               //calculate crystal orbiting in mm (amplitude-related to crystal center)
               //----------------------------------------------------------------------
               IF ("PAR_MAIN".MCONST_DIA_CAL_P2 > 0.0)   THEN 
                   #xt_orb_mm := 0.5 * ((#max_val_ctr_x_pos - #min_val_ctr_x_pos) / "PAR_MAIN".MCONST_DIA_CAL_P2 * 100.0);     
               END_IF;     

               //set calculation done flag
               //-------------------------
               #orb_calc_done   :=  true;            

               //reset counter 
               //-------------
               #count_msr   :=  0;

           END_IF;

           //set phase related orbiting limit
           //--------------------------------
           IF ("APC".STATUS = "APC".NECK)  THEN
               #up_lim_xt_orb   :=  "PAR_MAIN".MCONST_XT_ORB_LIM_NE;
               #rst_lim_xt_orb  :=  "CNF".RST_LIM_XT_ORB_NE;
           ELSIF ("APC".STATUS = "APC".SHOULDER)  THEN
               #up_lim_xt_orb   :=  "PAR_MAIN".MCONST_XT_ORB_LIM_SH;
               #rst_lim_xt_orb  :=  "CNF".RST_LIM_XT_ORB_SH;
           ELSE 
               #up_lim_xt_orb   :=  "PAR_MAIN".MCONST_XT_ORB_LIM_BY;
               #rst_lim_xt_orb  :=  "CNF".RST_LIM_XT_ORB_BY;
           END_IF;

           //evaluate crystal orbiting
           //-------------------------
           IF #orb_calc_done THEN
               //set orbiting alarm
               //------------------
               IF (#xt_orb_mm > #up_lim_xt_orb) OR "FLT".XT_ORB_ABV_LIM  THEN
                   IF (#set_flt <= 10) THEN      //ten consecutive calculations above limit
                       #set_flt := #set_flt + 1;

                   ELSE
                       //set alarm message
                       //-----------------
                       "FLT".XT_ORB_ABV_LIM  :=  TRUE;

                       //reset orbiting alarm
                       //--------------------
                       IF (#xt_orb_mm < #rst_lim_xt_orb)  THEN
                           IF (#reset_flt <= 30) THEN   //thirty consecutive calculations below limit
                               #reset_flt := #reset_flt + 1;

                           ELSE
                               //reset alarm message and flags
                               //-----------------------------
                               "FLT".XT_ORB_ABV_LIM  :=  FALSE;
                               #set_flt             :=  0;
                               #reset_flt           :=  0;
                           END_IF;
                       ELSE 
                           #reset_flt := 0;
                       END_IF;
                   END_IF;
               ELSE
                   #set_flt := 0;
               END_IF;
           END_IF;

       //crystal orbiting is deactivated
       //-------------------------------                          
       ELSE
           "FLT".XT_ORB_ABV_LIM  :=  FALSE;
           #xt_orb_mm           :=  0.0;
           #count_msr           :=  0;
           #set_flt             :=  0;
           #reset_flt           :=  0;
       END_IF;

       //set display value crystal orbiting
       //----------------------------------
       "DIS".ACT_XT_ORB  :=  #xt_orb_mm;
END_FUNCTION_BLOCK

FUNCTION_BLOCK "BM_MLT_LVL_MON"   // FB93, SCL
{ S7_Optimized_Access := 'FALSE' }
VERSION : 0.0
// --------------------------------------------------------------------------------
//     program     :    BM_MLT_LVL_MON
//     description :    melt level monitoring       
//     name        :    G. Eibelsh鋟ser
//     date        :    28.10.2009
// 
//     revision    :
//     name        :
//     date        :    
//                     (c)PVATepla AG
//     --------------------------------------------------------------------------------
   VAR
      ctl_mlt_drift_on : Bool;
      ctl_mlt_drift_on_dly : Int;
      cal_mlt_lvl_mm : Real;
      ini_mlt_lvl_mm : Real;
   END_VAR
BEGIN


       //monitoring of melt level in phases IDLE and BODY
       //------------------------------------------------
       IF ("APC".STATUS = "APC".IDLE) OR ("APC".STATUS = "APC".BODY) THEN 
           //calibrate melt level in unit mm
           //-------------------------------
           #cal_mlt_lvl_mm  :=  "AV".AVG_PRD_2_CTR_Y * "PAR_MAIN".MCONST_MLT_LVL_CAL;   //cal factor in unit mm/pixel

           //camera is on and circle sensor is selected
           //------------------------------------------
           IF "LT".CAM_ISP_ON AND ("AV".ACT_DVT_PRD_NO = 2.0) THEN 

               //automatic reset of melt level value in phase BODY
               //-------------------------------------------------
               IF ("APC".STATUS = "APC".BODY) AND ("AV".ACT_XT_LEN < "PAR_MAIN".BY_XT_LGH_MLT_LVL_RST) THEN     //actual crystal length below or equal activation length
                   "AV".ACT_MLT_LVL      :=  0.0;
                   #ini_mlt_lvl_mm      :=  #cal_mlt_lvl_mm;
                   #ctl_mlt_drift_on    :=  false;                          //disable melt drift control loop

               //melt level calculation
               //----------------------
               ELSE                                                        
                   IF ("APC".AUTOMATIC AND ("APC".STATUS = "APC".BODY) AND (REAL_TO_INT("PAR_MAIN".BY_CTL_MLT_DRIFT_ON) = 1) AND NOT "SY".CTL_OFFS_SPEED_ON) THEN  //crystal length exceeded activation length
                       #ctl_mlt_drift_on    :=  true;                       //enable melt drift control loop
                   ELSE
                       #ctl_mlt_drift_on    :=  false;                      //disable melt drift control loop
                   END_IF;

                   //stereo camera mode active
                   //-------------------------
                   IF (("CNF".ACT_DVC_CNF AND 2#0000_0000_0000_1000_0000_0000_0000_0000) = 2#0000_0000_0000_1000_0000_0000_0000_0000) THEN 
                       "AV".ACT_MLT_LVL   :=  "AV".S_CAM_AVG_MLT_LVL_CHG;  //pos. value >> melt gap gets larger, neg. value >> melt gap gets smaller

                   //single camera mode active
                   //-------------------------
                   ELSE 
                       //manual reset of melt level value
                       //--------------------------------
                       IF      NOT "APC".AUTOMATIC               //manual mode
                           OR      "SY".CTL_CR_SPD_COF_SMI       //semi mode crucible speed coeffizient
                           OR      "SY".CTL_MLT_LVL_SMI THEN     //semi mode crucible speed

                           IF "KYD".RST_MLT_LVL THEN
                               #ctl_mlt_drift_on    :=  false;                  //disable melt drift control loop while reseting 
                               #ini_mlt_lvl_mm      :=  #cal_mlt_lvl_mm;
                               "LT".RST_MLT_LVL      :=  TRUE;
                           END_IF;                
                       END_IF;
                       //calculation of actual melt level
                       //--------------------------------
                       "AV".ACT_MLT_LVL   :=  #cal_mlt_lvl_mm - #ini_mlt_lvl_mm;   //pos. value >> melt gap gets larger, neg. value >> melt gap gets smaller
                   END_IF;
               END_IF;

               //alarm setting in phase BODY
               //---------------------------
               IF ("APC".STATUS = "APC".BODY) AND ("PAR_MAIN".LIM_MLT_LVL_DEV >= 0.1) THEN   
                   //set alarm messages when distance from melt to funnel is too large
                   //-----------------------------------------------------------------
                   IF ("AV".ACT_MLT_LVL < "PAR_MAIN".LIM_MLT_LVL_DEV * 0.5) THEN
                       "FLT".DST_MLT_FNL_LRG :=  FALSE;

                   ELSIF ("AV".ACT_MLT_LVL > "PAR_MAIN".LIM_MLT_LVL_DEV) THEN
                       "FLT".DST_MLT_FNL_LRG :=  TRUE;

                   END_IF;

                   //set alarm messages when distance from melt to funnel is too small
                   //-----------------------------------------------------------------
                   IF ("AV".ACT_MLT_LVL > ("PAR_MAIN".LIM_MLT_LVL_DEV * (-0.5))) THEN  
                       "FLT".DST_MLT_FNL_SML :=  FALSE;

                   ELSIF ("AV".ACT_MLT_LVL < ("PAR_MAIN".LIM_MLT_LVL_DEV * (-1.0))) THEN  
                       "FLT".DST_MLT_FNL_SML :=  TRUE;

                   END_IF;

               ELSE
                   "FLT".DST_MLT_FNL_LRG :=  FALSE;
                   "FLT".DST_MLT_FNL_SML :=  FALSE;

               END_IF;

           //reset variables and alarms
           //--------------------------
           ELSE
               "AV".ACT_MLT_LVL      :=  0.0;
               #ini_mlt_lvl_mm      :=  #cal_mlt_lvl_mm;
               #ctl_mlt_drift_on    :=  false;                          //disable melt drift control loop
               "FLT".DST_MLT_FNL_LRG :=  FALSE;
               "FLT".DST_MLT_FNL_SML :=  FALSE;

           END_IF;

       ELSE
           //reset variables and alarms
           //--------------------------
           "AV".ACT_MLT_LVL      :=  0.0;
           #ctl_mlt_drift_on    :=  false;                          //disable melt drift control loop
           "FLT".DST_MLT_FNL_LRG :=  FALSE;
           "FLT".DST_MLT_FNL_SML :=  FALSE;

       END_IF;

       //enable control loop melt level drift
       //------------------------------------
       "DC".CTL_MLT_DRIFT_ON :=  "SysOndelay"( DIN     := #ctl_mlt_drift_on,
                                           SetTime := 30,                      // setp. time
                                           ActTime := #ctl_mlt_drift_on_dly,    // act. time
                                           Tick    := "SysTick1s");              // timebase (1s)

       //write display value of actual melt level
       //----------------------------------------
       "DIS".ACT_MLT_LVL  :=  "AV".ACT_MLT_LVL;
END_FUNCTION_BLOCK

FUNCTION_BLOCK "BM_MLT_VIB_MON"   // FB94, SCL
{ S7_Optimized_Access := 'FALSE' }
VERSION : 0.0
// --------------------------------------------------------------------------------
//     program     :    BM_MLT_VIB_MON
//     description :    melt vibration monitoring
//     name        :    G. Eibelsh鋟ser
//     date        :    01.09.2011
// 
//     revision    :
//     name        :
//     date        :    
//                     (c)PVA Tepla AG
//     --------------------------------------------------------------------------------
   VAR
      melt_vib_mon : Bool;
      store_mlt_vib_raw : Bool;
      cnt_msr : Int;
      cnt_msr_raw : Int;
      cnt_1s : Int;
      mlt_vib_dist : Array[1..300] of Real;
      mlt_vib_dist_raw : Array[1..100] of Real;
      min_mlt_vib_dist : Real;
      max_mlt_vib_dist : Real;
      mlt_vib_dist_pix : Real;
   END_VAR
   VAR CONSTANT
      amt_of_msr : Int := 10;
      amt_msr_raw : Int := 100;
   END_VAR
BEGIN


       //activate melt vibration monitoring
       //----------------------------------
       #melt_vib_mon := "LT".CAM_ISP_ON;

       //melt vibration monitoring is activated
       //--------------------------------------                          
       IF #melt_vib_mon  THEN

           //read sensor vibration distance
           //------------------------------  
           IF "DV".NEW_MSR_TEL_RECV THEN                         //new measurement telegram received
               #cnt_msr                 := #cnt_msr + 1;         //increase counter variable after each measurement
               #mlt_vib_dist[#cnt_msr]   := "AV".ACT_MLT_VIB_DIST; //store melt vibration distance in array variable
           END_IF;

           //evaluate measurement points
           //---------------------------
           IF (#cnt_msr >= #amt_of_msr) THEN

               //call min max detection
               //----------------------
               "CM_MIN_MAX"( record      := #mlt_vib_dist,
                           amt_of_val  := #amt_of_msr,
                           min_value   := #min_mlt_vib_dist, 
                           max_value   := #max_mlt_vib_dist);

               //calculate difference between min and max value
               //----------------------------------------------
               #mlt_vib_dist_pix := #max_mlt_vib_dist - #min_mlt_vib_dist;     

               //reset counter 
               //-------------
               #cnt_msr   :=  0;
           END_IF;    

           //store raw values of melt vibration sensor
           //-----------------------------------------
           IF "LT".MSR_MLT_VIB_ON THEN 
               IF #store_mlt_vib_raw THEN

                   //read sensor vibration distance
                   //------------------------------  
                   IF "DV".NEW_MSR_TEL_RECV THEN                                     //new measurement telegram received
                       #cnt_msr_raw                   := #cnt_msr_raw + 1;           //increase counter variable after each measurement
                       #mlt_vib_dist_raw[#cnt_msr_raw] := "AV".ACT_MLT_VIB_DIST;       //store melt vibration distance in array variable
                   END_IF;
                   //stop storage after selected amount of values
                   //--------------------------------------------
                   IF (#cnt_msr_raw >= #amt_msr_raw) THEN 
                       #store_mlt_vib_raw   :=  false;
                   END_IF;
               END_IF;

               //write raw values in display variables in 1 second intervall
               //-----------------------------------------------------------
               IF (#cnt_msr_raw >= 1) THEN 
                   IF "SysTick1s" THEN
                       IF (#cnt_1s >= #amt_msr_raw) THEN                         //stop writing after selected amount of seconds
                           "LT".MSR_MLT_VIB_ON   :=  FALSE;
                       ELSE
                           #cnt_1s              := #cnt_1s + 1;                  //increase 1 second counter
                           "DIS".ACT_MLT_VIB_RAW := #mlt_vib_dist_raw[#cnt_1s];    //write display value
                       END_IF;
                   END_IF;
               END_IF;

           //reset variables
           //---------------
           ELSE     
               #cnt_msr_raw         :=  0;
               #cnt_1s              :=  0;
               "DIS".ACT_MLT_VIB_RAW :=  0.0;
           END_IF;

           //activate storage of raw values from melt vibration sensor
           //---------------------------------------------------------
           IF "KYD".MSR_MLT_VIB_ON AND NOT "LT".MSR_MLT_VIB_ON THEN
               "LT".MSR_MLT_VIB_ON   :=  TRUE;
               #store_mlt_vib_raw   :=  true;
           END_IF;

       //reset variables
       //---------------
       ELSE    
           #cnt_msr             :=  0;
           #cnt_msr_raw         :=  0;
           #cnt_1s              :=  0;
           #mlt_vib_dist_pix    :=  0.0;
           "DIS".ACT_MLT_VIB_RAW :=  0.0;
           "LT".MSR_MLT_VIB_ON   :=  FALSE;
           #store_mlt_vib_raw   :=  false;
       END_IF;

       //write display value of actual melt vibration
       //--------------------------------------------
       "DIS".ACT_MLT_VIB :=  #mlt_vib_dist_pix;
END_FUNCTION_BLOCK

FUNCTION_BLOCK "BM_S_CAM_EVAL"   // FB99, SCL
{ S7_Optimized_Access := 'FALSE' }
VERSION : 0.0
// --------------------------------------------------------------------------------
//     program     :    BM_S_CAM_EVAL
//     description :    stereo camera evaluation  
//     name        :    G. Eibelsh鋟ser
//     date        :    20.08.2019
//        
//     revision    :   
//     name        :   
//     date        :   
//        
//                     (c)PVA Tepla AG
//     --------------------------------------------------------------------------------
   VAR
      s_cam_1_init_rad_pt : Real;
      s_cam_2_init_rad_pt : Real;
      s_cam_last_cf_dia : Real;
      s_cam_act_mlt_lvl_chg : Real;
      ini_mlt_lvl_inp : Real;
   END_VAR
   VAR_TEMP
      term_1 : Real;
      term_2 : Real;
      term_3 : Real;
      term_4 : Real;
      delta_x1 : Real;
      delta_x2 : Real;
      delta_r : Real;
      delta_h : Real;
   END_VAR
BEGIN


       //calculate trigonometric terms (angle in radiant)
       //------------------------------------------------
       #term_1  :=  SIN("CNF".PI * ("PAR_MAIN".MCONST_ANG_OF_PLX_SCAM - "CNF".S_CAM_ANG_BETA /2) /180);
       #term_2  :=  SIN("CNF".PI * ("PAR_MAIN".MCONST_ANG_OF_PLX_SCAM + "CNF".S_CAM_ANG_BETA /2) /180);
       #term_3  :=  COS("CNF".PI * ("PAR_MAIN".MCONST_ANG_OF_PLX_SCAM - "CNF".S_CAM_ANG_BETA /2) /180);
       #term_4  :=  COS("CNF".PI * ("PAR_MAIN".MCONST_ANG_OF_PLX_SCAM + "CNF".S_CAM_ANG_BETA /2) /180);

       //store initial radius point during circle fit
       //--------------------------------------------
       IF  NOT "DV".S_CAM_RAD_RT_ACTV   THEN
           #s_cam_1_init_rad_pt :=  "AV".S_CAM_1_AVG_RAD_PT;  
           #s_cam_2_init_rad_pt :=  "AV".S_CAM_2_AVG_RAD_PT;

       ELSE 
           //calculate radius from measured points of both cameras
           //-----------------------------------------------------
           #delta_x1 :=  #s_cam_1_init_rad_pt - "AV".S_CAM_1_AVG_RAD_PT;
           #delta_x2 :=  #s_cam_2_init_rad_pt - "AV".S_CAM_2_AVG_RAD_PT;

           //calculate radius of crystal from both camera inputs
           //--------------------------------------------------- 
           #delta_r := (#delta_x2 / #term_1 - #delta_x1 / #term_2) / (#term_3 / #term_1 - #term_4 / #term_2);

           //calculate melt level change from both camera inputs
           //--------------------------------------------------- 
           #delta_h := (#delta_x2 / #term_3 - #delta_x1 / #term_4) / (#term_1 / #term_3 - #term_2 / #term_4);

       END_IF;

       //write diameter and melt level variable
       //--------------------------------------
       //reset diamter and melt level change when camera off or diameter measuement mode not selected
       //--------------------------------------------------------------------------------------------
       IF NOT ("LT".CAM_ISP_ON AND "LT".CAM_DIA) THEN
           "AV".S_CAM_ACT_XT_DIA     :=  0.0;
           #s_cam_act_mlt_lvl_chg   :=  0.0;
       //radius point evaluation
       //-----------------------
       ELSIF "DV".S_CAM_RAD_RT_ACTV  THEN
           "AV".S_CAM_ACT_XT_DIA     :=  #s_cam_last_cf_dia + #delta_r * 2 / "PAR_MAIN".MCONST_CAL_RAD_PT_SCAM * 100 - "AC".XT_MENISCUS;   //unit of diameter calibration factor is pix/100mm
           //melt level change
           //-----------------
           #s_cam_act_mlt_lvl_chg   :=  #delta_h / "PAR_MAIN".MCONST_CAL_MLT_LVL_SCAM *(-1);   //unit of melt level calibration factor is pix/mm - neg. value >> reduced gap, pos. val. >> increased gap

       //circle fit evaluation
       //---------------------
       ELSE
           "AV".S_CAM_ACT_XT_DIA     :=  "AV".S_CAM_1_ACT_DIA_CF / "PAR_MAIN".MCONST_CAL_CF_SCAM * 100 - "AC".XT_MENISCUS;     //unit of diameter calibration factor is pix/100mm
           #s_cam_last_cf_dia       :=  "AV".S_CAM_ACT_XT_DIA + "AC".XT_MENISCUS;
           #s_cam_act_mlt_lvl_chg   :=  0.0;
       END_IF;

       //set point evaluation type - radius point detection or circle fit
       //----------------------------------------------------------------
       IF ("APC".STATUS <= "APC".NECK) THEN
           "DV".S_CAM_RAD_RT_ACTV   :=  FALSE;
       ELSIF ((("APC".STATUS = "APC".SHOULDER) AND ("AV".S_CAM_AVG_XT_DIA > "PAR_MAIN".MCONST_CF_TO_RAD_PT_SCAM)) OR ("APC".STATUS = "APC".BODY)) THEN
           "DV".S_CAM_RAD_RT_ACTV   :=  TRUE;
       END_IF;

       //manual reset of melt level value
       //--------------------------------
       IF ("KYD".RST_MLT_LVL AND NOT "LT".CTL_MLT_DRIFT_ON) THEN                   //melt drift control must be off
           "LT".RST_MLT_LVL := "KYD".RST_MLT_LVL AND NOT "LT".CTL_MLT_DRIFT_ON;      //reset in cm_loops
       END_IF;

       //melt level change calc in body after minimum length
       //---------------------------------------------------
       IF ("APC".STATUS = "APC".BODY) AND ("AV".ACT_XT_LEN >= "PAR_MAIN".BY_XT_LGH_MLT_LVL_RST) AND NOT "LT".RST_MLT_LVL THEN
           "AV".S_CAM_ACT_MLT_LVL_CHG    :=  #ini_mlt_lvl_inp - #s_cam_act_mlt_lvl_chg;
       //reset melt level change values
       //------------------------------
       ELSE
           #ini_mlt_lvl_inp             :=  #s_cam_act_mlt_lvl_chg;
           "AV".S_CAM_ACT_MLT_LVL_CHG    :=  0.0;
       END_IF;
END_FUNCTION_BLOCK

FUNCTION_BLOCK "BM_CALL_CAM"   // FB100, SCL
{ S7_Optimized_Access := 'FALSE' }
VERSION : 0.0
// --------------------------------------------------------------------------------
//     program     :    BM_CALL_CAM
//     description :    call camera modules 
//     name        :    G. Eibelsh鋟ser
//     date        :    03.05.2010
// 
//     revision    :    
//     name        :    
//     date        :    
//                     (c)PVA Tepla AG
//     --------------------------------------------------------------------------------
   VAR
      CAM_1_COM : "BM_CAM_COM";
      CAM_1_RSP : "BM_CAM_RSP";
      CAM_CONTROL : "BM_CAM_CONTROL";
      cam_1_req_msr : Bool;
      cam_1_send_req : Bool;
      cam_2_send_req : Bool;
      cam_1_send_done : Bool;
      cam_1_send_err : Bool;
      cam_1_recv_ndr : Bool;
      cam_1_recv_err : Bool;
      cam_1_eval_data : Bool;
      cam_1_data_str_recv : Bool;
      enb_dia_eval : Bool;
      no_ctr_fnd : Bool;
      wait_for_rsp : Bool;
      phase_shift : Bool;
      itl_cam_flt : Bool;
      xt_rot_cam_trg_prv : Bool;
      kyd_ext_acq_trg_busy : Bool;
      do_fac_shot_with_dly : Bool;
      sta_tme_trig_fac_shot : Bool;
      send_fac_shot_msg : Bool;
      cam_1_recv_len : Int;
      retval_blk : Int;
      i : Int;
      "m" : Int;
      n : Int;
      no_ctr_fnd_dly : Int;
      wait_for_rsp_dly : Int;
      itl_cam_flt_dly : Int;
      cam_no_ctr_fnd_dly : Int;
      mlt_amt_of_blobs : Int;
      apc_status : Int;
      dly_cnt : Int;
      acq_cnt : Int;
      next_fac_pic : Int;   // 0= fac1 1= fac2 2= fac3 3= fac4
      dly_fac_shot : Int;
      dly_cnt_fac_shot : DInt;   // added for single shot of facet
      cam_1_send_stat : Word;
      cam_1_recv_stat : Word;
      dip_int_on_line : Real;
      dia_cir_fit : Real;
      dia_cir_fit_old : Real;
      ctr_x_crd_cir_fit : Real;
      ctr_y_crd_cir_fit : Real;
      mlt_vib_dist : Real;
      dia_line_msr : Real;
      dia_pts_incl : Real;
      dia_cal_cir_fit : Real;
      dia_cal_pts_incl : Real;
      ctr_x_crd_cal_cir_fit : Real;
      ctr_y_crd_cal_cir_fit : Real;
      s_cam_delta_r : Real;   // added for stereo camera test
      s_cam_delta_h : Real;
      dia_circ_fit_x1 : Real;
      dia_circ_fit_x2 : Real;
      act_radius_x1 : Real;
      act_radius_x2 : Real;
      ctr_x_circ_fit_s_cam1 : Real;
      ctr_y_circ_fit_s_cam1 : Real;
      ctr_x_circ_fit_s_cam2 : Real;
      ctr_y_circ_fit_s_cam2 : Real;
      plc_to_sherlock : String[254];
   END_VAR
   VAR_TEMP
      rot_trg_acq_req : Bool;
      ms_btw_fct : Real;
   END_VAR
   VAR CONSTANT
      max_pix_intensity : Int := 255;
      amt_of_fct : Int := 4;   // amount of facettes
      min_xt_rot : Int := 2;   // minimum crystal rotation for external acqisition trigger
      time_base : Real := 60000.0;   // minute in ms
      time_trig_fac : DInt := 180000;   // all 3 min
   END_VAR
BEGIN


       //call camera control 
       //-------------------
       #CAM_CONTROL();

       //switch external acquisition trigger on/off
       //------------------------------------------
       IF "LT".XT_ROT_OFF OR ("KYA".SET_XT_ROT < #min_xt_rot) THEN 
           "LT".EXT_ACQ_TRG_ON   :=  FALSE;
       ELSE
           "SM_POS_EDGE"(input   :=  "KYD".EXT_ACQ_TRG,         //button external acquisiton trigger on/off
                       busy    :=  #kyd_ext_acq_trg_busy,
                       output  :=  "LT".EXT_ACQ_TRG_ON);
       END_IF;

       //calculate time between two facettes in ms
       //-----------------------------------------
       IF "LT".EXT_ACQ_TRG_ON THEN 
           #ms_btw_fct :=  #time_base / "KYA".SET_XT_ROT /#amt_of_fct;
       ELSE
           #ms_btw_fct :=  0.0;
       END_IF;

       //reset delay time with positive edge of rotation indexer
       //-------------------------------------------------------
       IF "PDI".XT_ROT_CAM_TRG AND NOT #xt_rot_cam_trg_prv OR NOT "LT".EXT_ACQ_TRG_ON THEN
           #dly_cnt     :=  0;
           #acq_cnt     :=  0;

       //increase delay time with cycle time of previous cycle
       //-----------------------------------------------------
       ELSE
           #dly_cnt :=  #dly_cnt + "SY".OB1_PREV_CYCLE;
       END_IF;

       //For the facet pic
       IF "LT".EXT_ACQ_TRG_ON AND "LT".CAM_ISP_ON THEN
           #dly_cnt_fac_shot:= #dly_cnt_fac_shot + "SY".OB1_PREV_CYCLE;
           IF #dly_cnt_fac_shot > #time_trig_fac THEN
               #next_fac_pic:= #next_fac_pic + 1;
               IF #next_fac_pic > 3 THEN
                   #next_fac_pic:=0;
               END_IF;
               #dly_cnt_fac_shot:=0;
               #do_fac_shot_with_dly:=TRUE;
           END_IF;

       ELSE
           #dly_cnt_fac_shot:= 0;
           #next_fac_pic:=-1;
           #do_fac_shot_with_dly:=FALSE;
           #sta_tme_trig_fac_shot:=FALSE;
           #send_fac_shot_msg:=FALSE;
       END_IF;

       //store status of rotation indexer of current cycle
       //-------------------------------------------------
       #xt_rot_cam_trg_prv  :=  "PDI".XT_ROT_CAM_TRG;

       //set rotation triggered acquisition request when delay time over
       //---------------------------------------------------------------
       IF ("LT".EXT_ACQ_TRG_ON AND (#dly_cnt >= (REAL_TO_INT("KYA".CAM_ACQ_DLY) + (#acq_cnt * #ms_btw_fct)))) THEN
           //When the fac should be shot after 3 min then look for the right fac and then do the pic
           IF #do_fac_shot_with_dly AND (#next_fac_pic = #acq_cnt) THEN
               #do_fac_shot_with_dly:=FALSE;
               #sta_tme_trig_fac_shot:=TRUE;
           END_IF;
           #rot_trg_acq_req :=  true;
           #acq_cnt         :=  #acq_cnt + 1;
       ELSE
           #rot_trg_acq_req := false;
       END_IF;

       //If the fac is been triggert by the area between the facettes a time of 1/2 the 1/4 rot time
       IF #sta_tme_trig_fac_shot THEN
           #dly_fac_shot:= #dly_fac_shot + "SY".OB1_PREV_CYCLE;
           IF #dly_fac_shot >= #ms_btw_fct/2 THEN
               #send_fac_shot_msg:=TRUE;
               #dly_fac_shot:=0;
               #sta_tme_trig_fac_shot:=FALSE;
           END_IF;
       END_IF;

       //set camera measurement request
       //------------------------------
       IF "LT".CAM_ISP_ON THEN
           IF "LT".EXT_ACQ_TRG_ON  THEN                  //external acquisition trigger active
               IF #rot_trg_acq_req THEN                 //triggered from rotation indexer, one acquisiton per rotation
                   #cam_1_req_msr :=  true;
               END_IF;
           ELSIF ("CNF".IMG_AQI_TRG = 100)  THEN
               IF "SysTick100ms" THEN                    //10Hz
                   #cam_1_req_msr :=  true;
               END_IF;
           ELSIF ("CNF".IMG_AQI_TRG = 200)  THEN
               IF "SysTick200ms" THEN                    //5Hz
                   #cam_1_req_msr :=  true;
               END_IF;
           ELSIF ("CNF".IMG_AQI_TRG = 500)  THEN
               IF "SysTick500ms" THEN                    //2Hz
                   #cam_1_req_msr :=  true;
               END_IF;
           ELSIF ("CNF".IMG_AQI_TRG = 1000)  THEN
               IF "SysTick1s" THEN                       //1Hz
                   #cam_1_req_msr :=  true;
               END_IF;
           END_IF;
       ELSE        
           #cam_1_req_msr :=  false;    //reset measurement request
       END_IF;

       //write send string
       //-----------------
       IF (#CAM_1_COM.O_SEND_STAT = 16#0000) AND NOT #wait_for_rsp   THEN       //no send task running and response on last request received

           //switch on image acquisition
           //---------------------------
           IF #CAM_CONTROL.O_ACQ_ON THEN
               #plc_to_sherlock             :=  'acq_on_';                          //set data 
               #cam_1_send_req              :=  true;                               //set send request
               #wait_for_rsp                :=  true;                               //wait for response
               #CAM_CONTROL.O_ACQ_ON        :=  FALSE;

           //switch off image acquisition
           //---------------------------
           ELSIF #CAM_CONTROL.O_ACQ_OFF THEN
               #plc_to_sherlock             :=  'acq_off';                          //set data 
               #cam_1_send_req              :=  true;                               //set send request
               #wait_for_rsp                :=  true;                               //wait for response
               #CAM_CONTROL.O_ACQ_OFF       :=  FALSE;

           //switch on relative threshold
           //----------------------------
           ELSIF #CAM_CONTROL.O_THR_REL_ON THEN
               #plc_to_sherlock             :=  'thr_rel';                          //set data 
               #cam_1_send_req              :=  true;                               //set send request
               #wait_for_rsp                :=  true;                               //wait for response
               #CAM_CONTROL.O_THR_REL_ON    :=  FALSE;

           //switch switch on absolute threshold
           //-----------------------------------
           ELSIF #CAM_CONTROL.O_THR_ABS_ON THEN
               #plc_to_sherlock             :=  'thr_abs';                          //set data 
               #cam_1_send_req              :=  true;                               //set send request
               #wait_for_rsp                :=  true;                               //wait for response
               #CAM_CONTROL.O_THR_ABS_ON    :=  FALSE;

           //switch on neck measurement mode for stereo cameras     - added for stereo camera test
           //--------------------------------------------------
           ELSIF #CAM_CONTROL.O_CF_EVAL THEN
               #plc_to_sherlock             :=  'cfit_ne';                          //set data 
               #cam_1_send_req              :=  true;                               //set send request
               #wait_for_rsp                :=  true;                               //wait for response
               #CAM_CONTROL.O_CF_EVAL       :=  FALSE;

           //switch off neck measurement mode for stereo cameras
           //---------------------------------------------------
           ELSIF #CAM_CONTROL.O_RAD_PT_EVAL THEN
               #plc_to_sherlock             :=  'pfit_sb';                          //set data 
               #cam_1_send_req              :=  true;                               //set send request
               #wait_for_rsp                :=  true;                               //wait for response
               #CAM_CONTROL.O_RAD_PT_EVAL   :=  FALSE;

           //ROI coordinate change is requested
           //----------------------------------
           ELSIF #CAM_CONTROL.O_NEW_ROI_CRD    THEN
               #plc_to_sherlock             BLKMOV  #CAM_CONTROL.O_ROI_CRD_STRG;         //set data 
               #cam_1_send_req              :=  true;                               //set send request
               #wait_for_rsp                :=  true;                               //wait for response
               #CAM_CONTROL.O_NEW_ROI_CRD   :=  FALSE;                              //reset flag new ROI coordinates

           //ROI threshold change is requested
           //---------------------------------
           ELSIF #CAM_CONTROL.O_NEW_ROI_THR  THEN                                   //set data
               #plc_to_sherlock             BLKMOV  #CAM_CONTROL.O_ROI_THR_STRG;
               #cam_1_send_req              :=  true;                               //set send request
               #wait_for_rsp                :=  true;                               //wait for response
               #CAM_CONTROL.O_NEW_ROI_THR   :=  FALSE;                              //reset flag new ROI coordinates

           //ROI threshold 2 change is requested
           //---------------------------------
           ELSIF #CAM_CONTROL.O_NEW_ROI_THR_2  THEN                                 //set data from camera 2
               #plc_to_sherlock             BLKMOV  #CAM_CONTROL.O_ROI_THR_STRG_2;
               #cam_1_send_req              :=  true;                               //set send request
               #wait_for_rsp                :=  true;                               //wait for response
               #CAM_CONTROL.O_NEW_ROI_THR_2 :=  FALSE;                              //reset flag new ROI coordinates

           //do a single pic of the facet    
           ELSIF #send_fac_shot_msg THEN
               CASE #next_fac_pic OF 
                   0:#plc_to_sherlock       :=  'pic_fac1';                          //set data                    
                   1:#plc_to_sherlock       :=  'pic_fac2';                          //set data 
                   2:#plc_to_sherlock       :=  'pic_fac3';                          //set data 
                   3:#plc_to_sherlock       :=  'pic_fac4';                          //set data 
               END_CASE;
               #cam_1_send_req              :=  true;                               //set send request
               #wait_for_rsp                :=  true;                               //wait for response
               #send_fac_shot_msg           :=  FALSE;                              //reset flag new ROI coordinates

           //cyclic measurement is requested
           //-------------------------------
           ELSIF #cam_1_req_msr THEN     
               //set plc command string
               //----------------------
               IF "LT".CAM_MLT THEN
                   #plc_to_sherlock    :='mlt_msr';        //melt detection measurement
               ELSIF "LT".CAM_DIP THEN
                   #plc_to_sherlock    :='dip_msr';        //dipping detection
               ELSIF "LT".CAM_DIA THEN
                   IF "LT".CAM_PRD_1_SEL THEN
                       #plc_to_sherlock    :='dia_rec';    //diameter measurement with rectangle ROI
                   ELSIF "LT".CAM_PRD_2_SEL THEN 
                       #plc_to_sherlock    :='dia_msr';    //diameter measurement with segmented circle ROI
                   END_IF;
               END_IF;

               #cam_1_send_req  :=  true;               //set send request
               #wait_for_rsp    :=  true;               //wait for response

               //reset measurement request
               //-------------------------
               #cam_1_req_msr       :=  false;          

           END_IF;    
       END_IF;

       //call TCP/IP communication of sherlock
       //-------------------------------------
       #CAM_1_COM  (IO_SEND_REQ         :=  #cam_1_send_req,
                   IO_DATA_STR_RECV    :=  #cam_1_data_str_recv,
                   I_SEND_CON_ID       :=  "CNF".CAM_1_CON_ID_SEND,
                   I_RECV_CON_ID       :=  "CNF".CAM_1_CON_ID_RECV,
                   I_CP_ADR            :=  "CNF".CP_LADDR,
                   I_DATA_STRING       BLKMOV  #plc_to_sherlock);

                   #cam_1_send_done     :=  #CAM_1_COM.O_SEND_DONE;
                   #cam_1_send_err      :=  #CAM_1_COM.O_SEND_ERR;
                   #cam_1_recv_ndr      :=  #CAM_1_COM.O_RECV_NDR;
                   #cam_1_recv_err      :=  #CAM_1_COM.O_RECV_ERR;
                   #cam_1_recv_len      :=  #CAM_1_COM.O_RECV_LEN;

                   #cam_1_send_stat     :=  #CAM_1_COM.O_SEND_STAT;
                   #cam_1_recv_stat     :=  #CAM_1_COM.O_RECV_STAT;

       "DV".NEW_MSR_TEL_RECV :=  FALSE;  //reset new measurement telegram variable            

       //move data from receive DB to data DB
       //------------------------------------
       IF #cam_1_data_str_recv THEN
           #retval_blk          :=  BLKMOV(SRCBLK:= "BM_CAM_RECV_DB", DSTBLK=> "BM_CAM_EVAL_DB");
           #cam_1_data_str_recv :=  false;
           #wait_for_rsp        :=  false;

           //call camera data response evaluation
           //------------------------------------
           #CAM_1_RSP(  I_CAM_RECV_LEN  :=  #cam_1_recv_len,
                       I_PLC_TO_CAM    BLKMOV  #plc_to_sherlock);

           //status of image acquisition
           //---------------------------            
           "LT".CAM_ISP_ON :=  #CAM_1_RSP.O_ACQ_IS_ON;            

           //response is melting telegram string
           //-----------------------------------
           IF (#CAM_1_RSP.O_RSP_STRG S_COMP 'mlt=')  THEN
               #mlt_amt_of_blobs    :=  REAL_TO_INT(#CAM_1_RSP.O_REAL_VALUE[0]);
               #dip_int_on_line     :=  0.0;
               #dia_cir_fit         :=  0.0;
               #dia_pts_incl        :=  0.0;
               #mlt_vib_dist        :=  0.0;
               #dia_line_msr        :=  0.0;

               "DV".NEW_MSR_TEL_RECV :=  TRUE;   //set new measurement telegram variable          
           //response is dipping telegram string
           //-----------------------------------
           ELSIF (#CAM_1_RSP.O_RSP_STRG S_COMP 'dip=')  THEN
               #mlt_amt_of_blobs    :=  0;
               #dip_int_on_line     :=  #CAM_1_RSP.O_REAL_VALUE[0] / #max_pix_intensity * 100.0;
               #dia_cir_fit         :=  0.0;
               #dia_pts_incl        :=  0.0;
               #mlt_vib_dist        :=  0.0;
               #dia_line_msr        :=  0.0;

               "DV".NEW_MSR_TEL_RECV :=  TRUE;   //set new measurement telegram variable          
           //response is diameter telegram string
           //-----------------------------------
           ELSIF (#CAM_1_RSP.O_RSP_STRG S_COMP 'dia=')  THEN
               #mlt_amt_of_blobs    :=  0;
               #dip_int_on_line     :=  0.0;

               //single or stereo mode
               //---------------------
               IF "LT".CAM_PRD_2_SEL THEN 
                   //single camera mode
                   //------------------
                   IF (("CNF".ACT_DVC_CNF AND 2#0000_0000_0000_0000_0000_0001_0000_0000) = 2#0000_0000_0000_0000_0000_0001_0000_0000) THEN    
                       #dia_cir_fit             :=  #CAM_1_RSP.O_REAL_VALUE[0] / "PAR_MAIN".MCONST_DIA_CAL_P2 * 100;
                       #dia_pts_incl            :=  #CAM_1_RSP.O_REAL_VALUE[1];
                       #mlt_vib_dist            :=  #CAM_1_RSP.O_REAL_VALUE[2];
                       #dia_line_msr            :=  0.0;
                       #ctr_x_crd_cir_fit       :=  #CAM_1_RSP.O_REAL_VALUE[3];
                       #ctr_y_crd_cir_fit       :=  #CAM_1_RSP.O_REAL_VALUE[4];
                   //stereo camera mode
                   //------------------
                   ELSE      
                       "AV".S_CAM_1_ACT_DIA_CF   :=  #CAM_1_RSP.O_REAL_VALUE[0];  //new: measured diameter of circle fit of stereo camera 1 - neck phase - unit is pixel
                       "AV".S_CAM_2_ACT_DIA_CF   :=  #CAM_1_RSP.O_REAL_VALUE[1];  //new: measured diameter of circle fit of stereo camera 2 - neck phase - unit is pixel
                       "AV".S_CAM_1_ACT_RAD_PT   :=  #CAM_1_RSP.O_REAL_VALUE[2];  //new: average radius point (x- coordinate) of stereo camera 1 - shoulder and body phase - unit is pixel
                       "AV".S_CAM_2_ACT_RAD_PT   :=  #CAM_1_RSP.O_REAL_VALUE[3];  //new: average radius point (x- coordinate) of stereo camera 2 - shoulder and body phase - unit is pixel
                       "AV".S_CAM_1_ACT_CF_CTR_X :=  #CAM_1_RSP.O_REAL_VALUE[4];  //new: x-coordinate of center of circle fit stereo camera 1
                       "AV".S_CAM_1_ACT_CF_CTR_Y :=  #CAM_1_RSP.O_REAL_VALUE[5];  //new: y-coordinate of center of circle fit stereo camera 1
                       "AV".S_CAM_2_ACT_CF_CTR_X :=  #CAM_1_RSP.O_REAL_VALUE[6];  //new: x-coordinate of center of circle fit stereo camera 2
                       "AV".S_CAM_2_ACT_CF_CTR_Y :=  #CAM_1_RSP.O_REAL_VALUE[7];  //new: y-coordinate of center of circle fit stereo camera 2
                   END_IF;
               //line sensor
               //-----------    
               ELSIF "LT".CAM_PRD_1_SEL THEN 
                   #dia_cir_fit         :=  #CAM_1_RSP.O_REAL_VALUE[0] / "PAR_MAIN".MCONST_DIA_CAL_P2 * 100;
                   #mlt_vib_dist        :=  #CAM_1_RSP.O_REAL_VALUE[1];
                   #dia_line_msr        :=  #CAM_1_RSP.O_REAL_VALUE[2] / "PAR_MAIN".MCONST_DIA_CAL_P1 * 100;          
                   #ctr_x_crd_cir_fit   :=  #CAM_1_RSP.O_REAL_VALUE[3];
                   #ctr_y_crd_cir_fit   :=  #CAM_1_RSP.O_REAL_VALUE[4];
               END_IF;

               "DV".NEW_MSR_TEL_RECV :=  TRUE;   //set new measurement telegram variable          
           END_IF;
       END_IF;

       //detect process phase shift
       //--------------------------
       IF ("APC".STATUS <> #apc_status) THEN
           #phase_shift :=  true;
       ELSE
           #phase_shift :=  false;
       END_IF;

       #apc_status  := "APC".STATUS;  //store phase status of current cycle

       //built camera interlock flag 
       //---------------------------
       #itl_cam_flt :=  "SysOffdelay"(DIN     := #phase_shift,         // input
                                   SetTime := 30,                  // delay time
                                   ActTime := #itl_cam_flt_dly,     // actual time value
                                   Tick    := "SysTick100ms");

       //set camera fault messages
       //-------------------------
       "FLT".CAM_DATA_RECV   :=  #CAM_1_RSP.O_RSP_FLT;                //generell response error - not expected telegramm received
       "FLT".CAM_ROI_OUTSIDE :=  #CAM_1_RSP.O_ROI_OUTSIDE_FLT;        //ROI outside frame

       IF "APC".AUTOMATIC    THEN 
           //no measureable contrast found
           //-----------------------------
           "FLT".CAM_NO_CTR_FND  :=  "SysOndelay" (DIN     := #CAM_1_RSP.O_COMMON_ERROR AND NOT #itl_cam_flt,    // fault input
                                               SetTime := 10,                                              // delay time
                                               ActTime := #cam_no_ctr_fnd_dly,                              // actual time value
                                               Tick    := "SysTick100ms");
       ELSE
           "FLT".CAM_NO_CTR_FND  :=  FALSE;
           #cam_no_ctr_fnd_dly  :=  0;
       END_IF;

       //set alarm message no data from camera received
       //----------------------------------------------
       "FLT".CAM_NDR_TOUT    :=  "SysOndelay" (DIN     := #wait_for_rsp,            // fault input
                                           SetTime := 10,                      // delay time
                                           ActTime := #wait_for_rsp_dly,        // actual time value
                                           Tick    := "SysTick100ms");  

       //abort crystal down controlled by camera in dipping phase
       //--------------------------------------------------------
       IF("APC".STATUS = "APC".DIPPING) THEN
           IF "DC".XT_LFT_DN AND "DC".XT_LFT_FST  THEN     //crystal down with fast speed
               IF "FLT".CAM_NDR_TOUT THEN
                   "DV".ARB_XT_DN_BY_CAM     := TRUE;    //set flag abort crystal down by camera 
                   "FLT".CAM_DI_XT_DN_ARB    := TRUE;    //set alarm message crystal down by camera aborted
               END_IF;
           END_IF;
       ELSE   
           "DV".ARB_XT_DN_BY_CAM     := FALSE;    //reset flag abort crystal down by camera 
           "FLT".CAM_DI_XT_DN_ARB    := FALSE;    //reset alarm message crystal down by camera aborted
       END_IF;

       //switch heater temperature or crucible rotation to semi automatic mode when camera failed
       //----------------------------------------------------------------------------------------
       IF "DC".CTL_GRW_RTE_ON THEN                           //growth control requested from auto mode
           IF "SY".CTL_GRW_RTE_ON THEN                       //growth control is on
               "FLT".CAM_HTR_1_IN_SMI        := FALSE;       //reset alarm message heater 1 in semi automatic 
               "FLT".CAM_CRUC_ROT_IN_SMI     := FALSE;       //reset alarm message crucible rotation in semi automatic

               IF "FLT".CAM_NDR_TOUT THEN
                   //shoulder growth control - crucible rotation control parameterized
                   //-----------------------------------------------------------------
                   IF ("PAR_MAIN".SH_CRUC_ROT_CTL_ON = 1.0) THEN   
                       "DV".CRUC_ROT_SMI               := TRUE;    //set flag growth control off - switch crucible rotation to semi mode
                       "FLT".CAM_CRUC_ROT_IN_SMI       := TRUE;    //set alarm message growth rate control off and crucible rotation in semi mode 
                   //shoulder growth control - standard configuration
                   //------------------------------------------------
                   ELSE 
                       "DV".HTR_1_SMI                := TRUE;    //set flag growth control off - switch heater temperature to semi mode
                       "FLT".CAM_HTR_1_IN_SMI        := TRUE;    //set alarm message growth rate control off and heater temperature in semi mode 
                   END_IF;
               END_IF;
           ELSE                                                //growth control is off
               "DV".HTR_1_SMI    := FALSE;                       //reset flag growth control off - switch heater temperature to semi mode
               "DV".CRUC_ROT_SMI := FALSE;                       //reset flag growth control off - switch crucible rotation to semi mode
           END_IF;
       ELSE
           "FLT".CAM_HTR_1_IN_SMI        := FALSE;       //reset alarm message heater 1 in semi automatic 
           "FLT".CAM_CRUC_ROT_IN_SMI     := FALSE;       //reset alarm message crucible rotation in semi automatic
           "DV".HTR_1_SMI                := FALSE;       //reset flag growth control off - switch heater temperature to semi mode
           "DV".CRUC_ROT_SMI             := FALSE;       //reset flag growth control off - switch crucible rotation to semi mode
       END_IF;

       //switch crystal lift to semi automatic mode when camera failed
       //-------------------------------------------------------------
       IF "DC".CTL_DIA_ON THEN                           //diameter control requeseted from auto mode
           IF "SY".CTL_DIA_ON THEN                       //diameter control is on
               "FLT".CAM_DIA_CTRL_OFF    := FALSE;       //reset alarm message 

               IF "FLT".CAM_NDR_TOUT THEN
                   "DV".XT_LFT_SMI           := TRUE;    //set flag dia control off - switch crystal lift to semi mode 
                   "FLT".CAM_DIA_CTRL_OFF    := TRUE;    //set alarm message 
               END_IF;
           ELSE                                        //dia control is off
               "DV".XT_LFT_SMI   := FALSE;               //reset flag dia control off
           END_IF;
       ELSE
           "FLT".CAM_DIA_CTRL_OFF    := FALSE;           //reset alarm message dia control off
           "DV".XT_LFT_SMI           := FALSE;           //reset flag dia control off
       END_IF;

       //set manual init request
       //-----------------------
       IF "FLT".CAM_NDR_TOUT THEN 
           IF "DV".CAM_INIT THEN
               #wait_for_rsp    :=  false;
           END_IF;
       END_IF;

       //evaluate junk detection sensor result
       //-------------------------------------
       IF "LT".CAM_ISP_ON AND "DV".CAM_MLT_CHK AND "LT".CAM_MLT THEN
           IF (#mlt_amt_of_blobs = 0) THEN  //amount of blobs = 0
               IF ("SysTick1s" AND (#i < 70)) THEN
                   #i := #i + 1;
               END_IF;
           ELSE 
               #i := 0;
           END_IF;

           IF (#i > 60) THEN    //delay setting of complete flag
               "DV".CAM_MELT_COMPLETE    :=  TRUE;
           ELSE                       
               "DV".CAM_MELT_COMPLETE    :=  FALSE;
           END_IF;
       ELSE 
           "DV".CAM_MELT_COMPLETE    :=  FALSE;
           #i                       :=  0;
       END_IF;

       //evaluate seed detection sensor result
       //-------------------------------------
       IF "LT".CAM_ISP_ON AND "LT".CAM_DIP THEN
           IF (#dip_int_on_line < 100.0) THEN  //bright area of sensor < 100.0 %
               "DV".CAM_DIP_COMPLETE :=  TRUE;
           ELSE                       
               "DV".CAM_DIP_COMPLETE :=  FALSE;
           END_IF;
       ELSE 
           "DV".CAM_DIP_COMPLETE :=  FALSE;
       END_IF;

       //enable evaluation of diameter signal
       //------------------------------------
       IF ("SY".CTL_DIA_ON OR ("SY".CTL_GRW_RTE_ON AND NOT "LT".SMI_HTR_1_ON)) AND "LT".CAM_ISP_ON THEN
           IF (#n > 3)  THEN
               #enb_dia_eval    :=  true;       //enable diameter evaluation delayed
           ELSE
               IF "SysTick1s"    THEN
                   #n   :=  #n + 1;
               END_IF;
           END_IF;
       ELSE
           #enb_dia_eval    :=  false;          //disable diameter evaluation
           #n   :=  0;
       END_IF;

       (*
       //do evaluation of diameter signal
       //--------------------------------         
       IF enb_dia_eval THEN    //check deviation of +/- 3mm        
           IF DV.NEW_MSR_TEL_RECV THEN 
               IF ((dia_cir_fit > (dia_cir_fit_old + 3.0)) OR (dia_cir_fit < (dia_cir_fit_old - 3.0))) THEN
                   IF (m >= 19)  THEN
                       FLT.CAM_MSR_INSTAB  :=  TRUE;       //fault message after twenty measurements
                       m                   :=  0;
                   ELSE
                       dia_cir_fit :=  dia_cir_fit_old;    //overwrite diameter with last valid diameter
                       m           :=  m + 1;
                   END_IF;
               ELSE
                   m                   :=  0;
                   FLT.CAM_MSR_INSTAB  :=  FALSE;
               END_IF;
           END_IF;
       ELSE
           m                   :=  0;
           FLT.CAM_MSR_INSTAB  :=  FALSE;
       END_IF;     
       *)

       //store last valid diameter
       //-------------------------
       #dia_cir_fit_old     :=  #dia_cir_fit;

       //set camera outputs related to measurement mode
       //----------------------------------------------
       IF NOT "LT".CAM_ISP_ON   THEN                                             //camera off
           "AV".INP_BLOBS        :=  0.0;
           "AV".INP_BGT_AREA     :=  0.0;  
           "AV".INP_XT_DIA       :=  0.0; 
           "AV".ACT_DIA_PTS_INCL :=  0.0; 
           "AV".ACT_MLT_VIB_DIST :=  0.0;
           "AV".ACT_PRD_2_CTR_X  :=  0.0;
           "AV".ACT_PRD_2_CTR_Y  :=  0.0;
           #no_ctr_fnd          :=  false;                                      //reset fault flag no contrast found

       ELSIF "LT".CAM_MLT   THEN                                                 //melting detection
           "AV".INP_BLOBS        :=  #mlt_amt_of_blobs;
           "AV".INP_BGT_AREA     :=  0.0;  
           "AV".INP_XT_DIA       :=  0.0; 
           "AV".ACT_DIA_PTS_INCL :=  0.0;
           "AV".ACT_MLT_VIB_DIST :=  #mlt_vib_dist;
           "AV".ACT_PRD_2_CTR_X  :=  0.0;
           "AV".ACT_PRD_2_CTR_Y  :=  0.0;
           #no_ctr_fnd          :=  false;                                      //reset fault flag no contrast found

       ELSIF "LT".CAM_DIP THEN                                                   //dipping detection
           "AV".INP_BLOBS        :=  0.0;
           "AV".INP_BGT_AREA     :=  #dip_int_on_line;  
           "AV".INP_XT_DIA       :=  0.0; 
           "AV".ACT_DIA_PTS_INCL :=  0.0;
           "AV".ACT_MLT_VIB_DIST :=  #mlt_vib_dist;
           "AV".ACT_PRD_2_CTR_X  :=  0.0;
           "AV".ACT_PRD_2_CTR_Y  :=  0.0;
           #no_ctr_fnd          :=  false;                                      //reset fault flag no contrast found

       ELSIF "LT".CAM_DIA THEN                                                   //diameter measurement
           "AV".INP_BLOBS        :=  0.0;
           "AV".INP_BGT_AREA     :=  0.0;  
           "AV".ACT_MLT_VIB_DIST :=  #mlt_vib_dist;

           //two point measurement with rectangle ROI
           //----------------------------------------        
           IF "LT".CAM_PRD_1_SEL AND (REAL_TO_INT("PAR_MAIN".MCONST_DIA_MSR_MTH) = 0) THEN                                                           //two point measurement
               "AV".INP_XT_DIA       :=  #dia_line_msr - "AC".XT_MENISCUS;      //write actual value diameter
               "AV".ACT_PRD_2_CTR_X  :=  0.0;
               "AV".ACT_PRD_2_CTR_Y  :=  0.0;

           //circle fit with seqmented circle or rectangle ROI
           //-------------------------------------------------
           ELSE
               IF "PAR_MAIN".CTL_DIA_COR_SEL = 0 THEN
                   "AV".INP_XT_DIA       :=  #dia_cir_fit - "AC".XT_MENISCUS;
                   "AV".INP_CAL_XT_DIA   :=  #dia_cal_cir_fit - "AC".XT_MENISCUS;

               ELSIF "PAR_MAIN".CTL_DIA_COR_SEL = 1 THEN // 1 = Corr. with melt lvl so the melt lvl is been used to correct the measured diameter 
                   "AV".INP_XT_DIA       :=  #dia_cir_fit - "AC".XT_MENISCUS + ("PAR_MAIN".MCONST_DIA_COR_MLT_LVL * "AV".ACT_MLT_LVL);               //write actual value diameter
                   "AV".INP_CAL_XT_DIA   :=  #dia_cal_cir_fit - "AC".XT_MENISCUS + ("PAR_MAIN".MCONST_DIA_COR_MLT_LVL * "AV".ACT_MLT_LVL);               //write actual value diameter
               ELSIF "PAR_MAIN".CTL_DIA_COR_SEL = 2 THEN // 1 = Corr. with gap offset size so the measured diameter can be correct by an offset
                   "AV".INP_XT_DIA       :=  #dia_cir_fit - "AC".XT_MENISCUS + ("PAR_MAIN".MCONST_DIA_COR_GAP_DEV * ((-1.0)*"DIS".ACT_MLT_GAP_OFFS));//write actual value diameter
                   "AV".INP_CAL_XT_DIA   :=  #dia_cal_cir_fit - "AC".XT_MENISCUS + ("PAR_MAIN".MCONST_DIA_COR_MLT_LVL * ((-1.0)*"DIS".ACT_MLT_GAP_OFFS)); //write actual value diameter
               ELSE
                   "PAR_MAIN".CTL_DIA_COR_SEL := 0;
                   "AV".INP_XT_DIA       :=  #dia_cir_fit - "AC".XT_MENISCUS;
                   "AV".INP_CAL_XT_DIA   :=  #dia_cal_cir_fit - "AC".XT_MENISCUS;
               END_IF; 

               "AV".ACT_DIA_PTS_INCL :=  #dia_pts_incl;
               "AV".ACT_PRD_2_CTR_X  :=  #ctr_x_crd_cir_fit;
               "AV".ACT_PRD_2_CTR_Y  :=  #ctr_y_crd_cir_fit;
           END_IF;
       END_IF;

       //set display values
       //------------------
       "DIS".ACT_AMT_BLOBS           :=  "AV".INP_BLOBS;   
       "DIS".ACT_PER_BGT_AREA        :=  "AV".INP_BGT_AREA;  
       "DIS".ACT_PRD_2_CTR_X         :=  "AV".ACT_PRD_2_CTR_X;
       "DIS".ACT_PRD_2_CTR_Y         :=  "AV".ACT_PRD_2_CTR_Y;
       "DIS".ACT_DIA_PTS_INCL        :=  "AV".ACT_DIA_PTS_INCL;
END_FUNCTION_BLOCK

FUNCTION_BLOCK "BM_CAM_COM"   // FB101, SCL
{ S7_Optimized_Access := 'FALSE' }
VERSION : 0.0
// --------------------------------------------------------------------------------
//     program     :    BM_CAM_COM
//     description :    TCP IP Communication with CP343   
//     name        :    G. Eibelsh鋟ser
//     date        :    03.05.2010
// 
//     revision    :
//     name        :
//     date        :    
//                     (c)PVA Tepla AG
//     --------------------------------------------------------------------------------
   VAR_INPUT
      I_SEND_CON_ID : Int;
      I_RECV_CON_ID : Int;
      I_CP_ADR : Word;
      I_DATA_STRING : String[254];
      Recv_DB : Struct
         Any_id : Byte;
         Recv_DataType : Byte;
         Recv_Lenght : Word;
         Recv_DB_Number : Word;
         Recv_Byte_Pointer : DWord;
      END_STRUCT;
      pAny_recv_db AT Recv_DB : ANY;
   END_VAR
   VAR_OUTPUT
      O_SEND_DONE : Bool;
      O_SEND_ERR : Bool;
      O_RECV_NDR : Bool;
      O_RECV_ERR : Bool;
      O_SEND_STAT : Word;
      O_RECV_STAT : Word;
      O_RECV_LEN : Int;
   END_VAR
   VAR_IN_OUT
      IO_SEND_REQ : Bool;
      IO_DATA_STR_RECV : Bool;
   END_VAR
   VAR
      size_of_buf : Byte;
      send_len : Int;
      state_cnt : Int;
      send_data : String[254];
   END_VAR
   VAR CONSTANT
      crlf : String := '$R$L';   // carriage return, line feed
   END_VAR
BEGIN


       //send_data
       //---------
       IF (#O_SEND_STAT = 16#0000)  THEN            // no task is running
           //add carriage return and line feed to input string
           //-------------------------------------------------
           #send_data    := CONCAT(IN1:= #I_DATA_STRING, IN2:= #crlf);

           //read length of data string
           //--------------------------
           #send_len    := LEN(IN:= #send_data);

       END_IF;

       //call AG_SEND
       //------------
       "AG_SEND"(    ACT     :=  #IO_SEND_REQ,
                   ID      :=  #I_SEND_CON_ID,
                   LADDR   :=  #I_CP_ADR,
                   SEND    :=  #send_data,
                   LEN     :=  #send_len,
                   DONE    =>  #O_SEND_DONE,
                   ERROR   =>  #O_SEND_ERR,
                   STATUS  =>  #O_SEND_STAT);

       //reset send request
       //------------------
       #IO_SEND_REQ     :=  FALSE;

       //built any pointer
       //----------------
       #Recv_DB.Any_id            := 16#10;
       #Recv_DB.Recv_DataType     := 16#2;
       #Recv_DB.Recv_Lenght       := #size_of_buf;
       #Recv_DB.Recv_DB_Number    := 16#281;                //DB number as hex code
       #Recv_DB.Recv_Byte_Pointer := DW#16#84000000;

       //call AG_RECV
       //------------
       "AG_RECV"(    ID      :=  #I_RECV_CON_ID,
                   LADDR   :=  #I_CP_ADR,
                   RECV    :=  #pAny_recv_db,
                   NDR     =>  #O_RECV_NDR,
                   ERROR   =>  #O_RECV_ERR,
                   STATUS  =>  #O_RECV_STAT,
                   LEN     =>  #O_RECV_LEN);

       //set flag data string received
       //-----------------------------
       IF (#O_RECV_NDR AND #state_cnt = 2)  THEN
           #IO_DATA_STR_RECV :=  TRUE;
       END_IF;

       //presetting of receive buffer size
       //---------------------------------     
       IF #O_RECV_NDR THEN 
           IF ("BM_CAM_RECV_DB".Data[0] = '!') THEN
               #state_cnt   :=  1;
           ELSIF ("BM_CAM_RECV_DB".Data[0] = BYTE_TO_CHAR(16#FF)) THEN
               #state_cnt   :=  2;
           ELSE 
               #state_cnt   :=  0;
           END_IF;
       END_IF;   

       CASE #state_cnt OF
           //read data bytewise
           //------------------    
           0:  #size_of_buf :=  16#1;       //search first character "!"

           //read two byte
           //-------------
           1:  #size_of_buf :=  16#2;       //read length of telegram string

           //read complete data lenght
           //-------------------------    
           2:  #size_of_buf     := CHAR_TO_BYTE("BM_CAM_RECV_DB".Data[1]);   //read telegram

       END_CASE;
END_FUNCTION_BLOCK

FUNCTION_BLOCK "BM_CAM_RSP"   // FB102, SCL
{ S7_Optimized_Access := 'FALSE' }
VERSION : 0.0
// --------------------------------------------------------------------------------
//     program     :    BM_CAM_RSP
//     description :    camera response
//     name        :    G. Eibelsh鋟ser
//     date        :    13.09.2010
// 
//     revision    :
//     name        :
//     date        :    
//                     (c)PVA Tepla AG
//     --------------------------------------------------------------------------------
   VAR_INPUT
      I_CAM_RECV_LEN : Int;
      I_PLC_TO_CAM : String[254];
   END_VAR
   VAR_OUTPUT
      O_RSP_FLT : Bool;
      O_ROI_OUTSIDE_FLT : Bool;
      O_COMMON_ERROR : Bool;
      O_ACQ_IS_ON : Bool;
      O_RSP_STRG : String[4];
      O_REAL_VALUE : Array[0..19] of Real;   // increased for stereo camera test
   END_VAR
   VAR
      CONV_DATA_CAM_1 : "CHAR_TO_DINT";
      read_data : Bool;
      i : Int;
      n : Int;
      rsp_strg : String[254];
      rsp_strg_int : String[254];
   END_VAR
   VAR CONSTANT
      acq_on : String := 'acq_on_';
      acq_off : String := 'acq_off';
      thr_abs : String := 'thr_abs';
      thr_rel : String := 'thr_rel';
      dia_msr : String := 'dia_msr';
      dip_msr : String := 'dip_msr';
      mlt_msr : String := 'mlt_msr';
      dia_thr : String := 'dia_thr';
      dia_crd : String := 'dia_crd';
      dip_thr : String := 'dip_thr';
      dip_crd : String := 'dip_crd';
      mlt_thr : String := 'mlt_thr';
      mlt_crd : String := 'mlt_crd';
      vib_thr : String := 'vib_thr';
      vib_crd : String := 'vib_crd';
      dia_rec : String := 'dia_rec';
      rec_thr : String := 'rec_thr';
      rec_crd : String := 'rec_crd';
      cfit_ne : String := 'cfit_ne';
      pfit_sb : String := 'pfit_sb';
      rke1_cc : String := 'rke1_cc';
      rke2_cc : String := 'rke2_cc';
      pic_fac1 : String := 'pic_fac1';
      pic_fac2 : String := 'pic_fac2';
      pic_fac3 : String := 'pic_fac3';
      pic_fac4 : String := 'pic_fac4';
   END_VAR
BEGIN


       //delete response string initially
       //--------------------------------
       #rsp_strg        := DELETE(IN:= #rsp_strg, L:= 254, P:= -1);

       //length of received string without CRLF
       //--------------------------------------
       #n   :=  #I_CAM_RECV_LEN - 2;

       //built response string from datablock bytes
       //------------------------------------------
       FOR #i := 1 TO #n DO 
           #rsp_strg := CONCAT(IN1:= #rsp_strg, IN2:= CHAR_TO_STRING("BM_CAM_EVAL_DB".Data[#i-1]));
       END_FOR;

       //isolate first seven bytes of PLC command
       //----------------------------------------
       #I_PLC_TO_CAM        := LEFT (IN:= #I_PLC_TO_CAM, L:= 7);
       #O_RSP_STRG          := 'init';  //initialise response output response string

       #O_RSP_FLT           := false;   //reset response fault
       #O_ROI_OUTSIDE_FLT   := false;   //reset ROI outside fault
       #O_COMMON_ERROR      := false;   //reset common error fault

       //acquisition on
       //--------------
       IF (#I_PLC_TO_CAM S_COMP #acq_on) THEN
           IF (#rsp_strg S_COMP 'acq_on_=ok') THEN
               #O_ACQ_IS_ON :=  true;
           ELSE
               #O_RSP_FLT   :=  true;
           END_IF;

       //acquisition off    
       //---------------
       ELSIF (#I_PLC_TO_CAM S_COMP #acq_off) THEN
           IF (#rsp_strg S_COMP 'acq_off=ok') THEN
               #O_ACQ_IS_ON :=  false;
           ELSE
               #O_RSP_FLT   :=  true;
           END_IF;

       //absolute threshold
       //------------------
       ELSIF (#I_PLC_TO_CAM S_COMP #thr_abs) THEN
           IF NOT (#rsp_strg S_COMP 'thr_abs=ok') THEN
               #O_RSP_FLT   :=  true;
           END_IF;

       //relative threshold
       //------------------
       ELSIF (#I_PLC_TO_CAM S_COMP #thr_rel) THEN
           IF NOT (#rsp_strg S_COMP 'thr_rel=ok') THEN
               #O_RSP_FLT   :=  true;
           END_IF;

       //neck measurement mode stereo cameras
       //------------------------------------
       ELSIF (#I_PLC_TO_CAM S_COMP #cfit_ne) THEN
           IF NOT (#rsp_strg S_COMP 'cfit_ne=ok') THEN
               #O_RSP_FLT   :=  true;
           END_IF;

       //shoulder body measurement mode stereo cameras
       //---------------------------------------------
       ELSIF (#I_PLC_TO_CAM S_COMP #pfit_sb) THEN
           IF NOT (#rsp_strg S_COMP 'pfit_sb=ok') THEN
               #O_RSP_FLT   :=  true;
           END_IF;

       //rake ROI stereo camera 1 coordinate change
       //------------------------------------------
       ELSIF (#I_PLC_TO_CAM S_COMP #rke1_cc) THEN
           IF NOT (#rsp_strg S_COMP 'rke1_cc=ok') THEN
               #O_RSP_FLT   :=  true;
           END_IF;

       //rake ROI stereo camera 2 coordinate change
       //------------------------------------------
       ELSIF (#I_PLC_TO_CAM S_COMP #rke2_cc) THEN
           IF NOT (#rsp_strg S_COMP 'rke2_cc=ok') THEN
               #O_RSP_FLT   :=  true;
           END_IF;

       //diameter threshold seqmented circle ROI
       //---------------------------------------
       ELSIF (#I_PLC_TO_CAM S_COMP #dia_thr) THEN
           IF NOT (#rsp_strg S_COMP 'dia_thr=ok') THEN
               #O_RSP_FLT   :=  true;
           END_IF;

       //diameter threshold rectangle ROI
       //--------------------------------
       ELSIF (#I_PLC_TO_CAM S_COMP #rec_thr) THEN
           IF NOT (#rsp_strg S_COMP 'rec_thr=ok') THEN
               #O_RSP_FLT   :=  true;
           END_IF;

       //diameter seqmented circle ROI coordinates
       //-----------------------------------------
       ELSIF (#I_PLC_TO_CAM S_COMP #dia_crd) THEN
           IF NOT(#rsp_strg S_COMP 'dia_crd=ok') THEN
               #O_RSP_FLT   :=  true;
           END_IF;

       //diameter rectangle ROI coordinates
       //----------------------------------
       ELSIF (#I_PLC_TO_CAM S_COMP #rec_crd) THEN
           IF NOT(#rsp_strg S_COMP 'rec_crd=ok') THEN
               #O_RSP_FLT   :=  true;
           END_IF;

       //melt vibration threshold
       //------------------------
       ELSIF (#I_PLC_TO_CAM S_COMP #vib_thr) THEN
           IF NOT (#rsp_strg S_COMP 'vib_thr=ok') THEN
               #O_RSP_FLT   :=  true;
           END_IF;

       //melt vibration ROI coordinates
       //------------------------------
       ELSIF (#I_PLC_TO_CAM S_COMP #vib_crd) THEN
           IF NOT(#rsp_strg S_COMP 'vib_crd=ok') THEN
               #O_RSP_FLT   :=  true;
           END_IF;

       //NEW with stereo cam
       ELSIF #I_PLC_TO_CAM S_COMP #pic_fac1 OR 
           #I_PLC_TO_CAM S_COMP #pic_fac2 OR 
           #I_PLC_TO_CAM S_COMP #pic_fac3 OR 
           #I_PLC_TO_CAM S_COMP #pic_fac4 THEN
           IF NOT ((#rsp_strg S_COMP 'pic_fac1=ok')OR
            (#rsp_strg S_COMP 'pic_fac2=ok') OR
            (#rsp_strg S_COMP 'pic_fac3=ok') OR
            (#rsp_strg S_COMP 'pic_fac4=ok'))THEN
               #O_RSP_FLT   :=  true;
           END_IF;

       //diameter measurement with seqmented circle ROI
       //----------------------------------------------
       ELSIF (#I_PLC_TO_CAM S_COMP #dia_msr) THEN
           #rsp_strg_int    := LEFT (IN:= #rsp_strg, L:= 4);         //isolate first four bytes of response string
           IF (#rsp_strg_int S_COMP 'dia=') THEN
               #O_RSP_STRG  BLKMOV  #rsp_strg_int;
               #read_data   :=  true;
           ELSE
               #rsp_strg_int    := LEFT (IN:= #rsp_strg, L:= 17);    //isolate first seventeen bytes of response string  
               IF (#rsp_strg_int S_COMP 'exe_err=ROIoutsde') THEN        //execution error= ROI outside 
                   #O_ROI_OUTSIDE_FLT   :=  true;
               ELSIF (#rsp_strg_int S_COMP 'exe_err=Commn err') THEN     //execution error= common error
                   #O_COMMON_ERROR  :=  true;
               ELSE
                   ;
                   //O_RSP_FLT   :=  true;
               END_IF;
           END_IF;

       //diameter measurement with rectangle ROI
       //---------------------------------------
       ELSIF (#I_PLC_TO_CAM S_COMP #dia_rec) THEN
           #rsp_strg_int    := LEFT (IN:= #rsp_strg, L:= 4);         //isolate first four bytes of response string
           IF (#rsp_strg_int S_COMP 'dia=') THEN
               #O_RSP_STRG  BLKMOV  #rsp_strg_int;
               #read_data   :=  true;
           ELSE
               #rsp_strg_int    := LEFT (IN:= #rsp_strg, L:= 17);    //isolate first seventeen bytes of response string  
               IF (#rsp_strg_int S_COMP 'exe_err=ROIoutsde') THEN        //execution error= ROI outside 
                   #O_ROI_OUTSIDE_FLT   :=  true;
               ELSIF (#rsp_strg_int S_COMP 'exe_err=Commn err') THEN     //execution error= common error
                   #O_COMMON_ERROR  :=  true;
               ELSE
                   ;
                   //O_RSP_FLT   :=  true;
               END_IF;
           END_IF;


      //dipping threshold
      //-----------------
       ELSIF (#I_PLC_TO_CAM S_COMP #dip_thr) THEN
           IF NOT (#rsp_strg S_COMP 'dip_thr=ok') THEN
               #O_RSP_FLT   :=  true;
           END_IF;

      //dipping ROI coordinates
      //-----------------------
       ELSIF (#I_PLC_TO_CAM S_COMP #dip_crd) THEN
           IF NOT (#rsp_strg S_COMP 'dip_crd=ok') THEN
               #O_RSP_FLT   :=  true;
           END_IF;

      //dipping measurement
      //-------------------
      ELSIF (#I_PLC_TO_CAM S_COMP #dip_msr) THEN
           #rsp_strg_int    := LEFT (IN:= #rsp_strg, L:= 4);         //isolate first four bytes of response string
           IF (#rsp_strg_int S_COMP 'dip=') THEN
               #O_RSP_STRG  BLKMOV  #rsp_strg_int;
               #read_data   :=  true;
           ELSE
               #rsp_strg_int    := LEFT (IN:= #rsp_strg, L:= 17);    //isolate first seventeen bytes of response string  
               IF (#rsp_strg_int S_COMP 'exe_err=ROIoutsde') THEN        //execution error= ROI outside 
                   #O_ROI_OUTSIDE_FLT   :=  true;
               ELSIF (#rsp_strg_int S_COMP 'exe_err=Commn err') THEN     //execution error= common error
                   #O_COMMON_ERROR  :=  true;
               ELSE
                   #O_RSP_FLT   :=  true;
               END_IF;
           END_IF;

       //melting threshold
       //-----------------
       ELSIF (#I_PLC_TO_CAM S_COMP #mlt_thr) THEN
           IF NOT (#rsp_strg S_COMP 'mlt_thr=ok') THEN
               #O_RSP_FLT   :=  true;
           END_IF;

      //melting ROI coordinates
      //-----------------------
       ELSIF (#I_PLC_TO_CAM S_COMP #mlt_crd) THEN
           IF NOT (#rsp_strg S_COMP 'mlt_crd=ok') THEN
               #O_RSP_FLT   :=  true;
           END_IF;

      //melting measurement
      //-------------------
       ELSIF (#I_PLC_TO_CAM S_COMP #mlt_msr) THEN
           #rsp_strg_int    := LEFT (IN:= #rsp_strg, L:= 4);         //isolate first four bytes of response string
           IF (#rsp_strg_int S_COMP 'mlt=') THEN
               #O_RSP_STRG  BLKMOV  #rsp_strg_int;
               #read_data   :=  true;
           ELSE
               #rsp_strg_int    := LEFT (IN:= #rsp_strg, L:= 17);    //isolate first seventeen bytes of response string  
               IF (#rsp_strg_int S_COMP 'exe_err=ROIoutsde') THEN        //execution error= ROI outside 
                   #O_ROI_OUTSIDE_FLT   :=  true;
               ELSIF (#rsp_strg_int S_COMP 'exe_err=Commn err') THEN     //execution error= common error
                   #O_COMMON_ERROR  :=  true;
               ELSE
                   #O_RSP_FLT   :=  true;
               END_IF;
           END_IF;
       END_IF;

       //response received, read data
       //----------------------------
       IF #read_data    THEN 

           //call conversion from character variables to double integer
           //----------------------------------------------------------
           #CONV_DATA_CAM_1(I_AMT_OF_BYTES   := #I_CAM_RECV_LEN);  

           //read output variables and scale
           //-------------------------------
           #O_REAL_VALUE[0]  := DINT_TO_REAL(#CONV_DATA_CAM_1.O_CAM_VALUE[0]) / 100;     
           #O_REAL_VALUE[1]  := DINT_TO_REAL(#CONV_DATA_CAM_1.O_CAM_VALUE[1]) / 100;     
           #O_REAL_VALUE[2]  := DINT_TO_REAL(#CONV_DATA_CAM_1.O_CAM_VALUE[2]) / 100;     
           #O_REAL_VALUE[3]  := DINT_TO_REAL(#CONV_DATA_CAM_1.O_CAM_VALUE[3]) / 100;     
           #O_REAL_VALUE[4]  := DINT_TO_REAL(#CONV_DATA_CAM_1.O_CAM_VALUE[4]) / 100;
           #O_REAL_VALUE[5]  := DINT_TO_REAL(#CONV_DATA_CAM_1.O_CAM_VALUE[5]) / 100;
           #O_REAL_VALUE[6]  := DINT_TO_REAL(#CONV_DATA_CAM_1.O_CAM_VALUE[6]) / 100;
           #O_REAL_VALUE[7]  := DINT_TO_REAL(#CONV_DATA_CAM_1.O_CAM_VALUE[7]) / 100;
           #O_REAL_VALUE[8]  := DINT_TO_REAL(#CONV_DATA_CAM_1.O_CAM_VALUE[8]) / 100;
           #O_REAL_VALUE[9]  := DINT_TO_REAL(#CONV_DATA_CAM_1.O_CAM_VALUE[9]) / 100;
           #O_REAL_VALUE[10] := DINT_TO_REAL(#CONV_DATA_CAM_1.O_CAM_VALUE[10]) / 100;        //added for stereo camera test
           #O_REAL_VALUE[11] := DINT_TO_REAL(#CONV_DATA_CAM_1.O_CAM_VALUE[11]) / 100;
           #O_REAL_VALUE[12] := DINT_TO_REAL(#CONV_DATA_CAM_1.O_CAM_VALUE[12]) / 100;
           #O_REAL_VALUE[13] := DINT_TO_REAL(#CONV_DATA_CAM_1.O_CAM_VALUE[13]) / 100;
           #O_REAL_VALUE[14] := DINT_TO_REAL(#CONV_DATA_CAM_1.O_CAM_VALUE[14]) / 100;
           #O_REAL_VALUE[15] := DINT_TO_REAL(#CONV_DATA_CAM_1.O_CAM_VALUE[15]) / 100;
           #O_REAL_VALUE[16] := DINT_TO_REAL(#CONV_DATA_CAM_1.O_CAM_VALUE[16]) / 100;
           #O_REAL_VALUE[17] := DINT_TO_REAL(#CONV_DATA_CAM_1.O_CAM_VALUE[17]) / 100;
           #O_REAL_VALUE[18] := DINT_TO_REAL(#CONV_DATA_CAM_1.O_CAM_VALUE[18]) / 100;
           #O_REAL_VALUE[19] := DINT_TO_REAL(#CONV_DATA_CAM_1.O_CAM_VALUE[19]) / 100;

           #read_data   :=  false;

       END_IF;
END_FUNCTION_BLOCK

FUNCTION_BLOCK "BM_CAM_CONTROL"   // FB103, SCL
{ S7_Optimized_Access := 'FALSE' }
VERSION : 0.0
// --------------------------------------------------------------------------------
//     program     :    BM_CAM_CONTROL
//     description :    camera acqisition and ROI control 
//     name        :    G. Eibelsh鋟ser
//     date        :    08.07.2010
// 
//     revision    :    melt vibration sensor in diameter measurement added
//     name        :    G. Eibelsh鋟ser
//     date        :    26.08.2011
//        
//     revision    :    GCL CGS1218 stereo camera 2. threshold
//     name        :    John Wang
//     date        :    04.08.2020
//        
//                     (c)PVA Tepla AG
//     --------------------------------------------------------------------------------
   VAR_OUTPUT
      O_ACQ_ON : Bool;
      O_ACQ_OFF : Bool;
      O_THR_REL_ON : Bool;
      O_THR_ABS_ON : Bool;
      O_NEW_ROI_CRD : Bool;
      O_NEW_ROI_THR : Bool;
      O_NEW_ROI_THR_2 : Bool;
      O_CF_EVAL : Bool;   // added for stereo camera test
      O_RAD_PT_EVAL : Bool;
      O_ROI_CRD_STRG : String[60];
      O_ROI_THR_STRG : String[20];
      O_ROI_THR_STRG_2 : String[20];
   END_VAR
   VAR
      new_roi_crd : Bool;
      new_thr_req : Bool;
      new_thr_req_2 : Bool;
      enb_set_params : Bool;
      new_mlt_vib_roi_crd : Bool;
      new_mlt_vib_thr_req : Bool;
      s_cam_rad_rt_actv_prv : Bool;
      set_params_dly : Int;
      apc_status_prv : Int;
      set_center_x : Real;
      set_center_y : Real;
      set_outer_radius : Real;
      set_inner_radius : Real;
      set_start_angle : Real;
      set_stop_angle : Real;
      set_width : Real;
      set_height : Real;
      ac_set_sen_thr : Real;
      ac_set_sen_thr_2 : Real;
      kya_set_sen_thr : Real;
      set_thr : Real;
      set_thr_2 : Real;
      center_x_old : Real;
      center_y_old : Real;
      start_angle_old : Real;
      stop_angle_old : Real;
      inner_radius_old : Real;
      outer_radius_old : Real;
      width_old : Real;
      height_old : Real;
      thr_old : Real;
      thr_old_2 : Real;
      set_mlt_vib_center_x : Real;
      set_mlt_vib_center_y : Real;
      set_mlt_vib_width : Real;
      set_mlt_vib_thr : Real;
      mlt_vib_center_x_old : Real;
      mlt_vib_center_y_old : Real;
      mlt_vib_width_old : Real;
      mlt_vib_thr_old : Real;
      set_ctr_x_scam_1 : Real;   // added for stereo camera test
      set_ctr_y_scam_1 : Real;
      set_width_scam_1 : Real;
      set_height_scam_1 : Real;
      set_ctr_x_scam_1_old : Real;
      set_ctr_y_scam_1_old : Real;
      set_width_scam_1_old : Real;
      set_height_scam_1_old : Real;
      set_ctr_x_scam_2 : Real;
      set_ctr_y_scam_2 : Real;
      set_width_scam_2 : Real;
      set_height_scam_2 : Real;
      set_ctr_x_scam_2_old : Real;
      set_ctr_y_scam_2_old : Real;
      set_width_scam_2_old : Real;
      set_height_scam_2_old : Real;
      center_x : String[7];
      center_y : String[7];
      start_angle : String[7];
      stop_angle : String[7];
      inner_radius : String[7];
      outer_radius : String[7];
      width : String[7];
      height : String[7];
      mlt_vib_center_x : String[7];
      mlt_vib_center_y : String[7];
      mlt_vib_width : String[7];
      roi_crd_strg : String[60];
      thr_cmd : String[8];
      thr_cmd_2 : String[8];
      thr : String[6];
      thr_2 : String[6];
      mlt_vib_thr : String[6];
      roi_thr_strg : String[20];
      roi_thr_strg_2 : String[20];
      ctr_x_scam1 : String[7];   // - added for stereo camera test
      ctr_y_scam1 : String[7];
      width_scam1 : String[7];
      height_scam1 : String[7];
      ctr_x_scam2 : String[7];
      ctr_y_scam2 : String[7];
      width_scam2 : String[7];
      height_scam2 : String[7];
   END_VAR
   VAR CONSTANT
      delimiter : Char := ';';
   END_VAR
BEGIN


       //selection of camera
       //-------------------
       IF "APC".AUTOMATIC    THEN                                    //automatic mode
           IF "DC".CAM_SEL_1 THEN
               "LT".CAM_SEL_1 := TRUE; 
               "LT".CAM_SEL_2 := FALSE;
           ELSIF  "DC".CAM_SEL_2 AND "CNF".CONF_CAM_2 THEN
               "LT".CAM_SEL_1 := FALSE;       
               "LT".CAM_SEL_2 := TRUE;
           ELSE
               "LT".CAM_SEL_1 := TRUE;                               //set camera 1 as default
               "LT".CAM_SEL_2 := FALSE;
           END_IF;

       ELSE                                                        //manual mode
           IF ("KYD".CAM_SEL_1 OR "LT".CAM_SEL_1) AND NOT "KYD".CAM_SEL_2 THEN
               "LT".CAM_SEL_1 := TRUE;
               "LT".CAM_SEL_2 := FALSE;
           ELSIF  ("KYD".CAM_SEL_2 OR "LT".CAM_SEL_2) AND "CNF".CONF_CAM_2 AND NOT "KYD".CAM_SEL_1 THEN
               "LT".CAM_SEL_1 := FALSE;       
               "LT".CAM_SEL_2 := TRUE;
           ELSE
               "LT".CAM_SEL_1 := TRUE;                               //set camera 1 as default
               "LT".CAM_SEL_2 := FALSE;
           END_IF;

       END_IF;

       //set camera control signals
       //--------------------------
       IF "APC".AUTOMATIC    THEN                                        //automatic mode
           "DV".CAM_ISP_ON   :=  "DC".CAM_ISP_ON;
       ELSE                                                            //manuell mode
           IF ("KYD".CAM_ISP_ON OR "LT".CAM_ISP_ON) AND NOT "KYD".CAM_ISP_OFF THEN
               "DV".CAM_ISP_ON   :=  TRUE;
           ELSE 
               "DV".CAM_ISP_ON   :=  FALSE;
           END_IF;
       END_IF;

       //set manual init request
       //-----------------------
       "DV".CAM_INIT :=  "KYD".CAM_INIT OR "DC".CAM_INIT;

       //initialize light variable diameter measurement after PLC restart
       //----------------------------------------------------------------
       IF ("SY".RUN_TIME < 3)    THEN
           "LT".CAM_DIA          :=  TRUE;       
           "STA".ACT_DVT_PRD_NO  :=  2.0;
       END_IF;

       //select measurement mode after inspection is on
       //----------------------------------------------
       IF "LT".CAM_ISP_ON AND "DV".CAM_ISP_ON  THEN
           IF "APC".AUTOMATIC    THEN                //automatic mode
               IF "DC".CAM_DIA  THEN
                   "LT".CAM_DIA  :=  TRUE;
                   "LT".CAM_DIP  :=  FALSE;
                   "LT".CAM_MLT  :=  FALSE;
                   "STA".ACT_DVT_PRD_NO  :=  2.0;
                   (*
                   //select ROI type phase related
                   //-----------------------------
                   IF (APC.STATUS = APC.NECK) THEN 
                       STA.ACT_DVT_PRD_NO  :=  REAL_TO_INT(PAR_MAIN.DIA_MSR_PRD_NE);    //set product number in phase neck   

                   ELSIF (APC.STATUS = APC.SHOULDER) THEN
                       STA.ACT_DVT_PRD_NO  :=  REAL_TO_INT(PAR_MAIN.DIA_MSR_PRD_SH);    //set product number in phase shoulder    

                   ELSIF (APC.STATUS = APC.BODY) THEN
                       STA.ACT_DVT_PRD_NO  :=  REAL_TO_INT(PAR_MAIN.DIA_MSR_PRD_BY);    //set product number in phase body   

                   END_IF; 
                   *)
               ELSIF "DC".CAM_DIP  THEN
                   "LT".CAM_DIA  :=  FALSE;
                   "LT".CAM_DIP  :=  TRUE;
                   "LT".CAM_MLT  :=  FALSE;
                   "STA".ACT_DVT_PRD_NO  :=  3.0;

               ELSIF "DC".CAM_MLT  THEN
                   "LT".CAM_DIA  :=  FALSE;
                   "LT".CAM_DIP  :=  FALSE;
                   "LT".CAM_MLT  :=  TRUE;
                   "STA".ACT_DVT_PRD_NO  :=  4.0;

               END_IF;
           ELSE                                    //manual mode
               IF "KYD".CAM_DIA  THEN
                   "LT".CAM_DIA  :=  TRUE;
                   "LT".CAM_DIP  :=  FALSE;
                   "LT".CAM_MLT  :=  FALSE;
                   "STA".ACT_DVT_PRD_NO  :=  2.0;

               ELSIF "KYD".CAM_DIP   THEN
                   "LT".CAM_DIA  :=  FALSE;
                   "LT".CAM_DIP  :=  TRUE;
                   "LT".CAM_MLT  :=  FALSE;
                   "STA".ACT_DVT_PRD_NO  :=  3.0;

               ELSIF "KYD".CAM_MLT   THEN
                   "LT".CAM_DIA  :=  FALSE;
                   "LT".CAM_DIP  :=  FALSE;
                   "LT".CAM_MLT  :=  TRUE;
                   "STA".ACT_DVT_PRD_NO  :=  4.0;

               END_IF;
               (* 
               //select ROI type of diameter measurement method
               //----------------------------------------------
               IF LT.CAM_DIA   THEN 
                   IF KYD.SEL_CAM_PRD_1 THEN           //set product 1
                       STA.ACT_DVT_PRD_NO    :=  1.0;

                   ELSIF KYD.SEL_CAM_PRD_2 THEN        //set product 2
                       STA.ACT_DVT_PRD_NO    :=  2.0;

                   ELSE    
                       IF LT.CAM_PRD_1_SEL THEN        
                           STA.ACT_DVT_PRD_NO :=  1.0;

                       ELSIF LT.CAM_PRD_2_SEL THEN
                           STA.ACT_DVT_PRD_NO :=  2.0;

                       END_IF;
                   END_IF;
               END_IF;
               *)
           END_IF;
       END_IF;

       //track light variables with camera measurement ROI type
       //------------------------------------------------------   
       IF ("STA".ACT_DVT_PRD_NO = 1.0) THEN
           "LT".CAM_PRD_1_SEL    :=  TRUE;
           "LT".CAM_PRD_2_SEL    :=  FALSE;
       ELSIF ("STA".ACT_DVT_PRD_NO = 2.0) THEN
           "LT".CAM_PRD_2_SEL    :=  TRUE;
           "LT".CAM_PRD_1_SEL    :=  FALSE;
       END_IF; 

       //copy status variable of actual DVT product number to AV value
       //-------------------------------------------------------------
       "AV".ACT_DVT_PRD_NO   :=  "STA".ACT_DVT_PRD_NO;         //historical reason

       //switch off/on image acquisition
       //-------------------------------
       IF "LT".CAM_ISP_ON THEN
           IF NOT "DV".CAM_ISP_ON THEN
               #O_ACQ_OFF   :=  TRUE;
           END_IF;
       ELSE
           IF "DV".CAM_ISP_ON THEN
               #O_ACQ_ON    :=  TRUE;
           ELSE
               #O_ACQ_ON    :=  FALSE;
           END_IF;
       END_IF;

       //set threshold type
       //------------------
       IF (("APC".STATUS = "APC".SHOULDER) AND (#apc_status_prv <> "APC".SHOULDER)) THEN              //phase switched to shoulder
           #O_THR_REL_ON    :=  FALSE;  
           #O_THR_ABS_ON    :=  TRUE;           //absolute threshold is active

       ELSIF   (("APC".STATUS <> "APC".SHOULDER) AND (#apc_status_prv = "APC".SHOULDER))    THEN      //phase switched from shoulder
           #O_THR_REL_ON    :=  TRUE;  
           #O_THR_ABS_ON    :=  FALSE;          //relative threshold is active
       END_IF;

       #apc_status_prv  :=  "APC".STATUS; //store phase code of active phase

       //set type of measurement evaluation             - added for stereo camera test
       //----------------------------------
       IF ("DV".S_CAM_RAD_RT_ACTV AND NOT #s_cam_rad_rt_actv_prv) THEN
           #O_CF_EVAL       :=  FALSE;
           #O_RAD_PT_EVAL   :=  TRUE;
       ELSIF (#s_cam_rad_rt_actv_prv AND NOT "DV".S_CAM_RAD_RT_ACTV) THEN
           #O_CF_EVAL       :=  TRUE;
           #O_RAD_PT_EVAL   :=  FALSE;
       END_IF;

       #s_cam_rad_rt_actv_prv   :=  "DV".S_CAM_RAD_RT_ACTV;   //store state of measurement evaluation     

       //set delayed enable flag for ROI settings
       //----------------------------------------        
       #enb_set_params := "SysOndelay"(   DIN     := "LT".CAM_ISP_ON,
                                       SetTime := 10,                              // setp. time
                                       ActTime := #set_params_dly,                  // act. time
                                       Tick    := "SysTick100ms");

       //evaluation of ROI settings
       //--------------------------    
       IF #enb_set_params THEN
           //melting detection
           //-----------------
           IF "LT".CAM_MLT THEN
               #set_center_x    :=  "CM_INSELECT"(auto    :=    "APC".AUTOMATIC,        // area in x-dimension
                                               track   :=    TRUE,
                                               ac      :=    ROUND("AC".SET_SEN_CTR_X),
                                               kya     :=    "KYA".SET_SEN_CTR_X_P4);

               #set_center_y    :=  "CM_INSELECT"(auto    :=    "APC".AUTOMATIC,        //area in y-dimension
                                               track   :=    TRUE,
                                               ac      :=    ROUND("AC".SET_SEN_CTR_Y),
                                               kya     :=    "KYA".SET_SEN_CTR_Y_P4);

               #set_width       :=  "CM_INSELECT"(auto    :=    "APC".AUTOMATIC,            //sensor width
                                               track   :=    TRUE,
                                               ac      :=    ROUND("AC".SET_SEN_WDH),
                                               kya     :=    "KYA".SET_SEN_WDH_P4);

               #set_height       :=  "CM_INSELECT"(auto    :=   "APC".AUTOMATIC,            //sensor height
                                               track   :=    TRUE,
                                               ac      :=    ROUND("AC".SET_SEN_HGT),
                                               kya     :=    "KYA".SET_SEN_HGT_P4);

               //check if ROI coordinate change is requested
               //-------------------------------------------
               IF NOT #O_NEW_ROI_CRD  THEN
                   //melting detection
                   //-----------------
                   IF (#set_center_x <> #center_x_old)   OR
                       (#set_center_y <> #center_y_old)  OR
                       (#set_width <> #width_old)        OR
                       (#set_height <> #height_old)      THEN 

                       #new_roi_crd :=  true;

                       //convert parameter values in string variables
                       //-------------------------------------------- 
                       #center_x    :=  DINT_TO_STRING (IN:= REAL_TO_DINT(#set_center_x * 100));
                       #center_y    :=  DINT_TO_STRING (IN:= REAL_TO_DINT(#set_center_y * 100));    
                       #width       :=  DINT_TO_STRING (IN:= REAL_TO_DINT(#set_width * 100));
                       #height      :=  DINT_TO_STRING (IN:= REAL_TO_DINT(#set_height * 100));    

                   END_IF;
               END_IF;

               //evaluate new ROI coordinate command string
               //------------------------------------------
               IF #new_roi_crd THEN

                   //delete ROI coordinate string
                   //----------------------------   
                   #roi_crd_strg := DELETE(IN:= #roi_crd_strg, L:= 60, P:= 0);

                   //built new ROI coordinate string
                   //-------------------------------     
                   #roi_crd_strg    := CONCAT(IN1:= 'mlt_crd=' , IN2:= #center_x);

                   #roi_crd_strg    := CONCAT(IN1:= #roi_crd_strg, IN2:= #delimiter);

                   #roi_crd_strg    := CONCAT(IN1:= #roi_crd_strg, IN2:= #center_y);

                   #roi_crd_strg    := CONCAT(IN1:= #roi_crd_strg, IN2:= #delimiter);

                   #roi_crd_strg    := CONCAT(IN1:= #roi_crd_strg, IN2:= #width);

                   #roi_crd_strg    := CONCAT(IN1:= #roi_crd_strg, IN2:= #delimiter);

                   #roi_crd_strg    := CONCAT(IN1:= #roi_crd_strg, IN2:= #height);

                   #O_ROI_CRD_STRG  :=  #roi_crd_strg;    //write new ROI coordinate string
                   #O_NEW_ROI_CRD   :=  true;

                   //save last requested ROI coordinates
                   //-----------------------------------
                   #center_x_old    :=  #set_center_x;
                   #center_y_old    :=  #set_center_y;
                   #width_old       :=  #set_width;
                   #height_old      :=  #set_height;

               END_IF;

           //dipping detection
           //-----------------    
           ELSIF "LT".CAM_DIP THEN
               #set_center_x    :=  "CM_INSELECT"(auto    :=    "APC".AUTOMATIC,            // area in x-dimension
                                               track   :=    TRUE,
                                               ac      :=    ROUND("AC".SET_SEN_CTR_X),
                                               kya     :=    "KYA".SET_SEN_CTR_X_P3);

               #set_center_y    :=  "CM_INSELECT"(auto    :=    "APC".AUTOMATIC,            //area in y-dimension
                                               track   :=    TRUE,
                                               ac      :=    ROUND("AC".SET_SEN_CTR_Y),
                                               kya     :=    "KYA".SET_SEN_CTR_Y_P3);

               #set_width       :=  "CM_INSELECT"(auto    :=    "APC".AUTOMATIC,            //sensor width
                                               track   :=    TRUE,
                                               ac      :=    ROUND("AC".SET_SEN_WDH),
                                               kya     :=    "KYA".SET_SEN_WDH_P3);

               //check if ROI coordinate change is requested
               //-------------------------------------------
               IF NOT #O_NEW_ROI_CRD  THEN
                   //dipping detection
                   //-----------------
                   IF (#set_center_x <> #center_x_old)           OR
                       (#set_center_y <> #center_y_old)          OR
                       (#set_width <> #width_old)                THEN 

                       #new_roi_crd :=  true;

                       //convert parameter values in string variables
                       //-------------------------------------------- 
                       #center_x    :=  DINT_TO_STRING (IN:= REAL_TO_DINT(#set_center_x * 100));
                       #center_y    :=  DINT_TO_STRING (IN:= REAL_TO_DINT(#set_center_y * 100));    
                       #width       :=  DINT_TO_STRING (IN:= REAL_TO_DINT(#set_width * 100));

                   END_IF;
               END_IF;

               //evaluate new ROI coordinate command string
               //------------------------------------------
               IF #new_roi_crd THEN

                   //delete ROI coordinate string
                   //----------------------------   
                   #roi_crd_strg := DELETE(IN:= #roi_crd_strg, L:= 60, P:= 0);

                   //built new ROI coordinate string
                   //-------------------------------     
                   #roi_crd_strg    := CONCAT(IN1:= 'dip_crd=' , IN2:= #center_x);

                   #roi_crd_strg    := CONCAT(IN1:= #roi_crd_strg, IN2:= #delimiter);

                   #roi_crd_strg    := CONCAT(IN1:= #roi_crd_strg, IN2:= #center_y);

                   #roi_crd_strg    := CONCAT(IN1:= #roi_crd_strg, IN2:= #delimiter);

                   #roi_crd_strg    := CONCAT(IN1:= #roi_crd_strg, IN2:= #width);

                   #O_ROI_CRD_STRG  :=  #roi_crd_strg;    //write new ROI coordinate string
                   #O_NEW_ROI_CRD   :=  true;

                   //save last requested ROI coordinates
                   //-----------------------------------
                   #center_x_old    :=  #set_center_x;
                   #center_y_old    :=  #set_center_y;
                   #width_old       :=  #set_width;

               END_IF;

           //diameter measurement
           //--------------------
           ELSIF "LT".CAM_DIA THEN
               //seqmented circle ROI is selected
               //--------------------------------
               IF "LT".CAM_PRD_2_SEL THEN 
                   //single camera mode
                   //------------------
                   IF (("CNF".ACT_DVC_CNF AND 2#0000_0000_0000_0000_0000_0001_0000_0000) = 2#0000_0000_0000_0000_0000_0001_0000_0000) THEN    
                       //read settings of circle sensor from recipe or manual input 
                       //----------------------------------------------------------
                       #set_center_x        :=  "CM_INSELECT"(auto    :=    "APC".AUTOMATIC,            //center of circle
                                                           track   :=    TRUE,
                                                           ac      :=    ROUND("AC".SET_SEN_CTR_X),
                                                           kya     :=    "KYA".SET_SEN_CTR_X_P2);

                       #set_center_y        :=  "CM_INSELECT"(auto    :=    "APC".AUTOMATIC,            //center of circle
                                                           track   :=    TRUE,
                                                           ac      :=    ROUND("AC".SET_SEN_CTR_Y),
                                                           kya     :=    "KYA".SET_SEN_CTR_Y_P2);

                       #set_start_angle    :=  "CM_INSELECT"( auto    :=    "APC".AUTOMATIC,            //seqment start angle
                                                           track   :=    TRUE,
                                                           ac      :=    ROUND("AC".SET_SEN_SEQ_STR_AGL),
                                                           kya     :=    "KYA".SET_SEN_SEQ_STR_AGL_P2);

                       #set_stop_angle      :=  "CM_INSELECT"(auto    :=    "APC".AUTOMATIC,            //seqment stop angle
                                                           track   :=    TRUE,
                                                           ac      :=    ROUND("AC".SET_SEN_SEQ_STP_AGL),
                                                           kya     :=    "KYA".SET_SEN_SEQ_STP_AGL_P2);

                       #set_inner_radius    :=  "CM_INSELECT"(auto    :=    "APC".AUTOMATIC,            //diameter of inner circle
                                                           track   :=    TRUE,
                                                           ac      :=    ROUND("AC".SET_SEN_IN_RAD),
                                                           kya     :=    "KYA".SET_SEN_IN_RAD_P2);

                       #set_outer_radius    :=  "CM_INSELECT"(auto    :=    "APC".AUTOMATIC,            //diameter of outer circle
                                                           track   :=    TRUE,
                                                           ac      :=    ROUND("AC".SET_SEN_OUT_RAD),
                                                           kya     :=    "KYA".SET_SEN_OUT_RAD_P2);

                       //check if ROI coordinate change is requested
                       //-------------------------------------------
                       IF NOT #O_NEW_ROI_CRD  THEN
                           //diameter measurement
                           //--------------------
                           IF  (#set_center_x <> #center_x_old)          OR
                               (#set_center_y <> #center_y_old)          OR
                               (#set_start_angle <> #start_angle_old)    OR
                               (#set_stop_angle <> #stop_angle_old)      OR 
                               (#set_inner_radius <> #inner_radius_old)  OR
                               (#set_outer_radius <> #outer_radius_old)  THEN

                               #new_roi_crd :=  true;

                               //convert parameter values in string variables
                               //-------------------------------------------- 
                               #center_x        :=  DINT_TO_STRING    (IN:= REAL_TO_DINT(#set_center_x * 100));
                               #center_y        :=  DINT_TO_STRING    (IN:= REAL_TO_DINT(#set_center_y * 100));    
                               #start_angle     :=  DINT_TO_STRING    (IN:= REAL_TO_DINT(#set_start_angle * 100));
                               #stop_angle      :=  DINT_TO_STRING    (IN:= REAL_TO_DINT(#set_stop_angle * 100));
                               #inner_radius    :=  DINT_TO_STRING    (IN:= REAL_TO_DINT(#set_inner_radius * 100));    
                               #outer_radius    :=  DINT_TO_STRING    (IN:= REAL_TO_DINT(#set_outer_radius * 100));

                           END_IF;

                           //evaluate new circle sensor ROI coordinate command string
                           //--------------------------------------------------------
                           IF #new_roi_crd THEN

                               //delete ROI coordinate string
                               //----------------------------   
                               #roi_crd_strg := DELETE(IN:= #roi_crd_strg, L:= 60, P:= 0);

                               //built new ROI coordinate string
                               //-------------------------------     
                               #roi_crd_strg    := CONCAT(IN1:= 'dia_crd=' , IN2:= #center_x);

                               #roi_crd_strg    := CONCAT(IN1:= #roi_crd_strg, IN2:= #delimiter);

                               #roi_crd_strg    := CONCAT(IN1:= #roi_crd_strg, IN2:= #center_y);

                               #roi_crd_strg    := CONCAT(IN1:= #roi_crd_strg, IN2:= #delimiter);

                               #roi_crd_strg    := CONCAT(IN1:= #roi_crd_strg, IN2:= #start_angle);

                               #roi_crd_strg    := CONCAT(IN1:= #roi_crd_strg, IN2:= #delimiter);

                               #roi_crd_strg    := CONCAT(IN1:= #roi_crd_strg, IN2:= #stop_angle);

                               #roi_crd_strg    := CONCAT(IN1:= #roi_crd_strg, IN2:= #delimiter);

                               #roi_crd_strg    := CONCAT(IN1:= #roi_crd_strg, IN2:= #inner_radius);

                               #roi_crd_strg    := CONCAT(IN1:= #roi_crd_strg, IN2:= #delimiter);

                               #roi_crd_strg    := CONCAT(IN1:= #roi_crd_strg, IN2:= #outer_radius);


                               #O_ROI_CRD_STRG      :=  #roi_crd_strg;    //write new ROI coordinate string
                               #O_NEW_ROI_CRD       :=  true;

